LIN {X 0,Y 157.711,Z 411.935,A -85,B 0,C 180,E1 -26136.375,E2 -26136.375} C_VEL
LIN {X 0,Y 161.502,Z 421.422,A -85,B 0,C 180,E1 -26138.842,E2 -26138.842} C_VEL
LIN {X 0,Y 167.93,Z 439.932,A -85,B 0,C 180,E1 -26142.847,E2 -26142.847} C_VEL
LIN {X 0,Y 172.068,Z 451.148,A -85,B 0,C 180,E1 -26145.625,E2 -26145.625} C_VEL
LIN {X 0,Y 176.253,Z 461.302,A -85,B 0,C 180,E1 -26148.517,E2 -26148.517} C_VEL
LIN {X 0,Y 181.026,Z 471.361,A -85,B 0,C 180,E1 -26151.736,E2 -26151.736} C_VEL
LIN {X 0,Y 187.397,Z 481.909,A -85,B 0,C 180,E1 -26155.593,E2 -26155.593} C_VEL
LIN {X 0,Y 193.568,Z 490.168,A -85,B 0,C 180,E1 -26158.913,E2 -26158.913} C_VEL
LIN {X 0,Y 201.708,Z 498.817,A -85,B 0,C 180,E1 -26162.732,E2 -26162.732} C_VEL
LIN {X 0,Y 208.546,Z 504.564,A -85,B 0,C 180,E1 -26165.489,E2 -26165.489} C_VEL
LIN {X 0,Y 218.387,Z 511.229,A -85,B 0,C 180,E1 -26168.946,E2 -26168.946} C_VEL
LIN {X 0,Y 231.636,Z 518.165,A -85,B 0,C 180,E1 -26172.885,E2 -26172.885} C_VEL
LIN {X 0,Y 242.773,Z 523.047,A -85,B 0,C 180,E1 -26175.876,E2 -26175.876} C_VEL
LIN {X 0,Y 253.89,Z 527.504,A -85,B 0,C 180,E1 -26178.827,E2 -26178.827} C_VEL
LIN {X 0,Y 260.167,Z 530.069,A -85,B 0,C 180,E1 -26180.673,E2 -26180.673} C_VEL
LIN {X 0,Y 265.407,Z 532.174,A -85,B 0,C 180,E1 -26182.392,E2 -26182.392} C_VEL
LIN {X 0,Y 269.507,Z 533.855,A -85,B 0,C 180,E1 -26184.013,E2 -26184.013} C_VEL
LIN {X 0,Y 272.328,Z 535.154,A -85,B 0,C 180,E1 -26185.56,E2 -26185.56} C_VEL
LIN {X 0,Y 274.967,Z 536.076,A -85,B 0,C 180,E1 -26187.07,E2 -26187.07} C_VEL
LIN {X 0,Y 276.582,Z 536.626,A -85,B 0,C 180,E1 -26188.544,E2 -26188.544} C_VEL
LIN {X 0,Y 277.498,Z 536.802,A -85,B 0,C 180,E1 -26190,E2 -26190} C_VEL
LIN {X 0,Y 276.603,Z 536.625,A -85,B 0,C 180,E1 -26191.456,E2 -26191.456} C_VEL
LIN {X 0,Y 274.515,Z 535.937,A -85,B 0,C 180,E1 -26193.198,E2 -26193.198} C_VEL
LIN {X 0,Y 272.324,Z 535.154,A -85,B 0,C 180,E1 -26194.44,E2 -26194.44} C_VEL
LIN {X 0,Y 268.7,Z 533.534,A -85,B 0,C 180,E1 -26196.334,E2 -26196.334} C_VEL
LIN {X 0,Y 265.444,Z 532.173,A -85,B 0,C 180,E1 -26197.607,E2 -26197.607} C_VEL
LIN {X 0,Y 260.186,Z 530.068,A -85,B 0,C 180,E1 -26199.327,E2 -26199.327} C_VEL
LIN {X 0,Y 251.348,Z 526.504,A -85,B 0,C 180,E1 -26201.867,E2 -26201.867} C_VEL
LIN {X 0,Y 239.951,Z 521.882,A -85,B 0,C 180,E1 -26204.866,E2 -26204.866} C_VEL
LIN {X 0,Y 226.976,Z 515.933,A -85,B 0,C 180,E1 -26208.439,E2 -26208.439} C_VEL
LIN {X 0,Y 213.38,Z 508.049,A -85,B 0,C 180,E1 -26212.749,E2 -26212.749} C_VEL
LIN {X 0,Y 202.925,Z 499.912,A -85,B 0,C 180,E1 -26216.758,E2 -26216.758} C_VEL
LIN {X 0,Y 195.267,Z 492.096,A -85,B 0,C 180,E1 -26220.256,E2 -26220.256} C_VEL
LIN {X 0,Y 187.81,Z 482.614,A -85,B 0,C 180,E1 -26224.146,E2 -26224.146} C_VEL
LIN {X 0,Y 181.961,Z 473.083,A -85,B 0,C 180,E1 -26227.651,E2 -26227.651} C_VEL
LIN {X 0,Y 177.726,Z 464.648,A -85,B 0,C 180,E1 -26230.43,E2 -26230.43} C_VEL
LIN {X 0,Y 173.629,Z 455.239,A -85,B 0,C 180,E1 -26233.234,E2 -26233.234} C_VEL
LIN {X 0,Y 169.867,Z 445.428,A -85,B 0,C 180,E1 -26235.824,E2 -26235.824} C_VEL
LIN {X 0,Y 166.21,Z 435.07,A -85,B 0,C 180,E1 -26238.245,E2 -26238.245} C_VEL
LIN {X 0,Y 161.21,Z 420.652,A -85,B 0,C 180,E1 -26241.342,E2 -26241.342} C_VEL
LIN {X 0,Y 157.598,Z 411.646,A -85,B 0,C 180,E1 -26243.703,E2 -26243.703} C_VEL
LIN {X 0,Y 153.19,Z 402.471,A -85,B 0,C 180,E1 -26246.795,E2 -26246.795} C_VEL
LIN {X 0,Y 148.612,Z 394.018,A -85,B 0,C 180,E1 -26250.424,E2 -26250.424} C_VEL
LIN {X 0,Y 144.236,Z 386.913,A -85,B 0,C 180,E1 -26254.476,E2 -26254.476} C_VEL
LIN {X 0,Y 141.463,Z 382.764,A -85,B 0,C 180,E1 -26257.501,E2 -26257.501} C_VEL
LIN {X 0,Y 138.857,Z 378.927,A -85,B 0,C 180,E1 -26260.878,E2 -26260.878} C_VEL
LIN {X 0,Y 136.291,Z 375.231,A -85,B 0,C 180,E1 -26265.06,E2 -26265.06} C_VEL
LIN {X 0,Y 135.757,Z 374.279,A -85,B 0,C 180,E1 -26266.149,E2 -26266.149} C_VEL
LIN {X 0,Y 133.455,Z 371.692,A -85,B 0,C 180,E1 -26272.056,E2 -26272.056} C_VEL
LIN {X 0,Y 132.719,Z 369.463,A -85,B 0,C 180,E1 -26276.586,E2 -26276.586} C_VEL
LIN {X 0,Y 132.574,Z 368.941,A -85,B 0,C 180,E1 -26280.002,E2 -26280.002} C_VEL
LIN {X 0,Y 132.851,Z 369.82,A -85,B 0,C 180,E1 -26284.173,E2 -26284.173} C_VEL
LIN {X 0,Y 135.292,Z 374.003,A -85,B 0,C 180,E1 -26292.566,E2 -26292.566} C_VEL
LIN {X 0,Y 136.12,Z 374.835,A -85,B 0,C 180,E1 -26294.198,E2 -26294.198} C_VEL
LIN {X 0,Y 138.416,Z 378.446,A -85,B 0,C 180,E1 -26298.121,E2 -26298.121} C_VEL
LIN {X 0,Y 139.473,Z 379.845,A -85,B 0,C 180,E1 -26299.599,E2 -26299.599} C_VEL
LIN {X 0,Y 142.528,Z 384.331,A -85,B 0,C 180,E1 -26303.331,E2 -26303.331} C_VEL
LIN {X 0,Y 145.453,Z 388.952,A -85,B 0,C 180,E1 -26306.356,E2 -26306.356} C_VEL
LIN {X 0,Y 147.78,Z 392.828,A -85,B 0,C 180,E1 -26308.495,E2 -26308.495} C_VEL
LIN {X 0,Y 151.379,Z 401.147,A -85,B 0,C 180,E1 -26311.635,E2 -26311.635} C_VEL
LIN {X 0,Y 155.437,Z 412.076,A -85,B 0,C 180,E1 -26314.84,E2 -26314.84} C_VEL
LIN {X 0,Y 156.568,Z 415.668,A -85,B 0,C 180,E1 -26315.702,E2 -26315.702} C_VEL
LIN {X 0,Y 154.129,Z 443.65,A -85,B 0,C 180,E1 -26316.777,E2 -26316.777} C_VEL
LIN {X 0,Y 152.023,Z 456.485,A -85,B 0,C 180,E1 -26317.57,E2 -26317.57} C_VEL
LIN {X 0,Y 148.735,Z 469.266,A -85,B 0,C 180,E1 -26318.773,E2 -26318.773} C_VEL
LIN {X 0,Y 145.582,Z 478.774,A -85,B 0,C 180,E1 -26319.973,E2 -26319.973} C_VEL
LIN {X 0,Y 141.897,Z 488.043,A -85,B 0,C 180,E1 -26321.487,E2 -26321.487} C_VEL
LIN {X 0,Y 137.778,Z 496.981,A -85,B 0,C 180,E1 -26323.375,E2 -26323.375} C_VEL
LIN {X 0,Y 133.274,Z 505.504,A -85,B 0,C 180,E1 -26325.677,E2 -26325.677} C_VEL
LIN {X 0,Y 129.051,Z 512.718,A -85,B 0,C 180,E1 -26328.156,E2 -26328.156} C_VEL
LIN {X 0,Y 125.096,Z 518.916,A -85,B 0,C 180,E1 -26330.801,E2 -26330.801} C_VEL
LIN {X 0,Y 120.577,Z 525.451,A -85,B 0,C 180,E1 -26334.349,E2 -26334.349} C_VEL
LIN {X 0,Y 115.984,Z 531.873,A -85,B 0,C 180,E1 -26339,E2 -26339} C_VEL
LIN {X 0,Y 111.97,Z 537.003,A -85,B 0,C 180,E1 -26343.937,E2 -26343.937} C_VEL
LIN {X 0,Y 108.806,Z 540.993,A -85,B 0,C 180,E1 -26349.191,E2 -26349.191} C_VEL
LIN {X 0,Y 106.705,Z 543.952,A -85,B 0,C 180,E1 -26354.725,E2 -26354.725} C_VEL
LIN {X 0,Y 105.264,Z 546.414,A -85,B 0,C 180,E1 -26362.326,E2 -26362.326} C_VEL
LIN {X 0,Y 105.047,Z 547.01,A -85,B 0,C 180,E1 -26366.164,E2 -26366.164} C_VEL
LIN {X 0,Y 105.171,Z 547.172,A -85,B 0,C 180,E1 -26370,E2 -26370} C_VEL
LIN {X 0,Y 105.038,Z 547.01,A -85,B 0,C 180,E1 -26373.836,E2 -26373.836} C_VEL
LIN {X 0,Y 105.226,Z 546.413,A -85,B 0,C 180,E1 -26377.676,E2 -26377.676} C_VEL
LIN {X 0,Y 106.705,Z 543.952,A -85,B 0,C 180,E1 -26385.275,E2 -26385.275} C_VEL
LIN {X 0,Y 108.806,Z 540.993,A -85,B 0,C 180,E1 -26390.809,E2 -26390.809} C_VEL
LIN {X 0,Y 111.97,Z 537.003,A -85,B 0,C 180,E1 -26396.063,E2 -26396.063} C_VEL
LIN {X 0,Y 115.99,Z 531.874,A -85,B 0,C 180,E1 -26400.999,E2 -26400.999} C_VEL
LIN {X 0,Y 120.636,Z 525.453,A -85,B 0,C 180,E1 -26405.631,E2 -26405.631} C_VEL
LIN {X 0,Y 126.046,Z 517.533,A -85,B 0,C 180,E1 -26409.881,E2 -26409.881} C_VEL
LIN {X 0,Y 131.142,Z 509.34,A -85,B 0,C 180,E1 -26413.099,E2 -26413.099} C_VEL
LIN {X 0,Y 136.063,Z 500.383,A -85,B 0,C 180,E1 -26415.78,E2 -26415.78} C_VEL
LIN {X 0,Y 140.126,Z 492.096,A -85,B 0,C 180,E1 -26417.711,E2 -26417.711} C_VEL
LIN {X 0,Y 144.306,Z 482.034,A -85,B 0,C 180,E1 -26419.548,E2 -26419.548} C_VEL
LIN {X 0,Y 147.764,Z 472.284,A -85,B 0,C 180,E1 -26420.881,E2 -26420.881} C_VEL
LIN {X 0,Y 150.284,Z 463.495,A -85,B 0,C 180,E1 -26421.833,E2 -26421.833} C_VEL
LIN {X 0,Y 152.647,Z 453.074,A -85,B 0,C 180,E1 -26422.656,E2 -26422.656} C_VEL
LIN {X 0,Y 154.169,Z 443.105,A -85,B 0,C 180,E1 -26423.25,E2 -26423.25} C_VEL
LIN {X 0,Y 156.565,Z 415.689,A -85,B 0,C 180,E1 -26424.298,E2 -26424.298} C_VEL
LIN {X 0,Y 153.862,Z 407.654,A -85,B 0,C 180,E1 -26426.368,E2 -26426.368} C_VEL
LIN {X 0,Y 149.993,Z 397.773,A -85,B 0,C 180,E1 -26429.538,E2 -26429.538} C_VEL
LIN {X 0,Y 147.077,Z 391.607,A -85,B 0,C 180,E1 -26432.133,E2 -26432.133} C_VEL
LIN {X 0,Y 143.786,Z 386.3,A -85,B 0,C 180,E1 -26435.312,E2 -26435.312} C_VEL
LIN {X 0,Y 141.521,Z 382.829,A -85,B 0,C 180,E1 -26437.819,E2 -26437.819} C_VEL
LIN {X 0,Y 139.084,Z 379.09,A -85,B 0,C 180,E1 -26440.966,E2 -26440.966} C_VEL
LIN {X 0,Y 138.007,Z 378.043,A -85,B 0,C 180,E1 -26442.468,E2 -26442.468} C_VEL
LIN {X 0,Y 136.91,Z 377.653,A -85,B 0,C 180,E1 -26444.037,E2 -26444.037} C_VEL
LIN {X 0,Y 133.217,Z 378.698,A -85,B 0,C 180,E1 -26450.653,E2 -26450.653} C_VEL
LIN {X 0,Y 132.394,Z 378.392,A -85,B 0,C 180,E1 -26453.213,E2 -26453.213} C_VEL
LIN {X 0,Y 132.218,Z 378.001,A -85,B 0,C 180,E1 -26454.058,E2 -26454.058} C_VEL
LIN {X 0,Y 131.788,Z 376.347,A -85,B 0,C 180,E1 -26457.706,E2 -26457.706} C_VEL
LIN {X 0,Y 131.702,Z 376.09,A -85,B 0,C 180,E1 -26460.763,E2 -26460.763} C_VEL
LIN {X 0,Y 131.924,Z 376.857,A -85,B 0,C 180,E1 -26464.199,E2 -26464.199} C_VEL
LIN {X 0,Y 134.158,Z 380.922,A -85,B 0,C 180,E1 -26472.444,E2 -26472.444} C_VEL
LIN {X 0,Y 134.823,Z 381.684,A -85,B 0,C 180,E1 -26473.853,E2 -26473.853} C_VEL
LIN {X 0,Y 137.252,Z 385.481,A -85,B 0,C 180,E1 -26478.181,E2 -26478.181} C_VEL
LIN {X 0,Y 140.462,Z 390.479,A -85,B 0,C 180,E1 -26482.523,E2 -26482.523} C_VEL
LIN {X 0,Y 143.478,Z 395.47,A -85,B 0,C 180,E1 -26485.863,E2 -26485.863} C_VEL
LIN {X 0,Y 147.492,Z 402.492,A -85,B 0,C 180,E1 -26489.626,E2 -26489.626} C_VEL
LIN {X 0,Y 152.1,Z 411.916,A -85,B 0,C 180,E1 -26493.375,E2 -26493.375} C_VEL
LIN {X 0,Y 156.129,Z 421.509,A -85,B 0,C 180,E1 -26496.312,E2 -26496.312} C_VEL
LIN {X 0,Y 159.764,Z 432.052,A -85,B 0,C 180,E1 -26498.817,E2 -26498.817} C_VEL
LIN {X 0,Y 163.355,Z 443.752,A -85,B 0,C 180,E1 -26501.513,E2 -26501.513} C_VEL
LIN {X 0,Y 166.675,Z 453.927,A -85,B 0,C 180,E1 -26504.209,E2 -26504.209} C_VEL
LIN {X 0,Y 170.416,Z 464.042,A -85,B 0,C 180,E1 -26507.268,E2 -26507.268} C_VEL
LIN {X 0,Y 174.817,Z 474.111,A -85,B 0,C 180,E1 -26510.702,E2 -26510.702} C_VEL
LIN {X 0,Y 178.982,Z 481.72,A -85,B 0,C 180,E1 -26513.606,E2 -26513.606} C_VEL
LIN {X 0,Y 184.846,Z 490.495,A -85,B 0,C 180,E1 -26517.285,E2 -26517.285} C_VEL
LIN {X 0,Y 190.862,Z 497.704,A -85,B 0,C 180,E1 -26520.58,E2 -26520.58} C_VEL
LIN {X 0,Y 198.504,Z 504.99,A -85,B 0,C 180,E1 -26524.206,E2 -26524.206} C_VEL
LIN {X 0,Y 208.801,Z 512.388,A -85,B 0,C 180,E1 -26528.27,E2 -26528.27} C_VEL
LIN {X 0,Y 221.304,Z 519.044,A -85,B 0,C 180,E1 -26532.307,E2 -26532.307} C_VEL
LIN {X 0,Y 235.113,Z 524.844,A -85,B 0,C 180,E1 -26536.165,E2 -26536.165} C_VEL
LIN {X 0,Y 246.769,Z 529.058,A -85,B 0,C 180,E1 -26539.279,E2 -26539.279} C_VEL
LIN {X 0,Y 255.571,Z 532.16,A -85,B 0,C 180,E1 -26541.871,E2 -26541.871} C_VEL
LIN {X 0,Y 261.478,Z 534.217,A -85,B 0,C 180,E1 -26543.97,E2 -26543.97} C_VEL
LIN {X 0,Y 264.483,Z 535.367,A -85,B 0,C 180,E1 -26545.428,E2 -26545.428} C_VEL
LIN {X 0,Y 267.412,Z 536.324,A -85,B 0,C 180,E1 -26547.058,E2 -26547.058} C_VEL
LIN {X 0,Y 269.258,Z 536.825,A -85,B 0,C 180,E1 -26548.504,E2 -26548.504} C_VEL
LIN {X 0,Y 270.33,Z 536.994,A -85,B 0,C 180,E1 -26550,E2 -26550} C_VEL
LIN {X 0,Y 269.274,Z 536.824,A -85,B 0,C 180,E1 -26551.496,E2 -26551.496} C_VEL
LIN {X 0,Y 267.267,Z 536.288,A -85,B 0,C 180,E1 -26553.015,E2 -26553.015} C_VEL
LIN {X 0,Y 264.455,Z 535.368,A -85,B 0,C 180,E1 -26554.573,E2 -26554.573} C_VEL
LIN {X 0,Y 261.075,Z 534.088,A -85,B 0,C 180,E1 -26556.181,E2 -26556.181} C_VEL
LIN {X 0,Y 255.574,Z 532.153,A -85,B 0,C 180,E1 -26558.134,E2 -26558.134} C_VEL
LIN {X 0,Y 246.768,Z 529.059,A -85,B 0,C 180,E1 -26560.72,E2 -26560.72} C_VEL
LIN {X 0,Y 235.074,Z 524.846,A -85,B 0,C 180,E1 -26563.838,E2 -26563.838} C_VEL
LIN {X 0,Y 221.304,Z 519.043,A -85,B 0,C 180,E1 -26567.693,E2 -26567.693} C_VEL
LIN {X 0,Y 208.846,Z 512.387,A -85,B 0,C 180,E1 -26571.725,E2 -26571.725} C_VEL
LIN {X 0,Y 200.755,Z 506.782,A -85,B 0,C 180,E1 -26574.84,E2 -26574.84} C_VEL
LIN {X 0,Y 192.265,Z 499.236,A -85,B 0,C 180,E1 -26578.686,E2 -26578.686} C_VEL
LIN {X 0,Y 185.303,Z 491.125,A -85,B 0,C 180,E1 -26582.438,E2 -26582.438} C_VEL
LIN {X 0,Y 179.655,Z 482.876,A -85,B 0,C 180,E1 -26585.929,E2 -26585.929} C_VEL
LIN {X 0,Y 174.806,Z 474.142,A -85,B 0,C 180,E1 -26589.293,E2 -26589.293} C_VEL
LIN {X 0,Y 170.971,Z 465.43,A -85,B 0,C 180,E1 -26592.278,E2 -26592.278} C_VEL
LIN {X 0,Y 168.022,Z 457.733,A -85,B 0,C 180,E1 -26594.68,E2 -26594.68} C_VEL
LIN {X 0,Y 164.732,Z 448.109,A -85,B 0,C 180,E1 -26597.371,E2 -26597.371} C_VEL
LIN {X 0,Y 161.357,Z 437.315,A -85,B 0,C 180,E1 -26600.028,E2 -26600.028} C_VEL
LIN {X 0,Y 157.158,Z 424.418,A -85,B 0,C 180,E1 -26602.959,E2 -26602.959} C_VEL
LIN {X 0,Y 153.804,Z 415.819,A -85,B 0,C 180,E1 -26605.35,E2 -26605.35} C_VEL
LIN {X 0,Y 150.072,Z 407.643,A -85,B 0,C 180,E1 -26608.208,E2 -26608.208} C_VEL
LIN {X 0,Y 146.074,Z 399.864,A -85,B 0,C 180,E1 -26611.642,E2 -26611.642} C_VEL
LIN {X 0,Y 142.005,Z 392.928,A -85,B 0,C 180,E1 -26615.709,E2 -26615.709} C_VEL
LIN {X 0,Y 139.441,Z 388.935,A -85,B 0,C 180,E1 -26618.738,E2 -26618.738} C_VEL
LIN {X 0,Y 137.25,Z 385.508,A -85,B 0,C 180,E1 -26621.817,E2 -26621.817} C_VEL
LIN {X 0,Y 134.783,Z 381.586,A -85,B 0,C 180,E1 -26626.239,E2 -26626.239} C_VEL
LIN {X 0,Y 131.818,Z 376.434,A -85,B 0,C 180,E1 -26636.945,E2 -26636.945} C_VEL
LIN {X 0,Y 131.715,Z 376.082,A -85,B 0,C 180,E1 -26640.766,E2 -26640.766} C_VEL
LIN {X 0,Y 131.953,Z 377.015,A -85,B 0,C 180,E1 -26644.106,E2 -26644.106} C_VEL
LIN {X 0,Y 134.175,Z 380.928,A -85,B 0,C 180,E1 -26652.096,E2 -26652.096} C_VEL
LIN {X 0,Y 134.866,Z 381.77,A -85,B 0,C 180,E1 -26653.564,E2 -26653.564} C_VEL
LIN {X 0,Y 137.314,Z 385.532,A -85,B 0,C 180,E1 -26657.886,E2 -26657.886} C_VEL
LIN {X 0,Y 140.622,Z 390.728,A -85,B 0,C 180,E1 -26662.329,E2 -26662.329} C_VEL
LIN {X 0,Y 144.3,Z 396.751,A -85,B 0,C 180,E1 -26666.291,E2 -26666.291} C_VEL
LIN {X 0,Y 147.272,Z 403.499,A -85,B 0,C 180,E1 -26669.188,E2 -26669.188} C_VEL
LIN {X 0,Y 151.416,Z 414.966,A -85,B 0,C 180,E1 -26672.854,E2 -26672.854} C_VEL
LIN {X 0,Y 152.317,Z 417.977,A -85,B 0,C 180,E1 -26673.622,E2 -26673.622} C_VEL
LIN {X 0,Y 150.023,Z 443.119,A -85,B 0,C 180,E1 -26674.584,E2 -26674.584} C_VEL
LIN {X 0,Y 147.77,Z 456.439,A -85,B 0,C 180,E1 -26675.399,E2 -26675.399} C_VEL
LIN {X 0,Y 144.404,Z 469.072,A -85,B 0,C 180,E1 -26676.581,E2 -26676.581} C_VEL
LIN {X 0,Y 141.129,Z 478.581,A -85,B 0,C 180,E1 -26677.765,E2 -26677.765} C_VEL
LIN {X 0,Y 137.284,Z 487.849,A -85,B 0,C 180,E1 -26679.26,E2 -26679.26} C_VEL
LIN {X 0,Y 133,Z 496.787,A -85,B 0,C 180,E1 -26681.151,E2 -26681.151} C_VEL
LIN {X 0,Y 128.289,Z 505.31,A -85,B 0,C 180,E1 -26683.46,E2 -26683.46} C_VEL
LIN {X 0,Y 123.824,Z 512.523,A -85,B 0,C 180,E1 -26685.951,E2 -26685.951} C_VEL
LIN {X 0,Y 119.659,Z 518.722,A -85,B 0,C 180,E1 -26688.644,E2 -26688.644} C_VEL
LIN {X 0,Y 114.846,Z 525.256,A -85,B 0,C 180,E1 -26692.27,E2 -26692.27} C_VEL
LIN {X 0,Y 109.942,Z 531.679,A -85,B 0,C 180,E1 -26697.088,E2 -26697.088} C_VEL
LIN {X 0,Y 105.604,Z 536.808,A -85,B 0,C 180,E1 -26702.235,E2 -26702.235} C_VEL
LIN {X 0,Y 102.183,Z 540.798,A -85,B 0,C 180,E1 -26707.773,E2 -26707.773} C_VEL
LIN {X 0,Y 99.83,Z 543.757,A -85,B 0,C 180,E1 -26713.645,E2 -26713.645} C_VEL
LIN {X 0,Y 98.213,Z 546.219,A -85,B 0,C 180,E1 -26721.772,E2 -26721.772} C_VEL
LIN {X 0,Y 97.952,Z 546.816,A -85,B 0,C 180,E1 -26725.886,E2 -26725.886} C_VEL
LIN {X 0,Y 98.077,Z 546.978,A -85,B 0,C 180,E1 -26730,E2 -26730} C_VEL
LIN {X 0,Y 97.944,Z 546.816,A -85,B 0,C 180,E1 -26734.115,E2 -26734.115} C_VEL
LIN {X 0,Y 98.183,Z 546.219,A -85,B 0,C 180,E1 -26738.231,E2 -26738.231} C_VEL
LIN {X 0,Y 99.83,Z 543.757,A -85,B 0,C 180,E1 -26746.355,E2 -26746.355} C_VEL
LIN {X 0,Y 102.183,Z 540.798,A -85,B 0,C 180,E1 -26752.227,E2 -26752.227} C_VEL
LIN {X 0,Y 105.603,Z 536.808,A -85,B 0,C 180,E1 -26757.765,E2 -26757.765} C_VEL
LIN {X 0,Y 109.953,Z 531.679,A -85,B 0,C 180,E1 -26762.908,E2 -26762.908} C_VEL
LIN {X 0,Y 114.085,Z 526.335,A -85,B 0,C 180,E1 -26766.99,E2 -26766.99} C_VEL
LIN {X 0,Y 118.657,Z 520.097,A -85,B 0,C 180,E1 -26770.656,E2 -26770.656} C_VEL
LIN {X 0,Y 122.787,Z 514.15,A -85,B 0,C 180,E1 -26773.38,E2 -26773.38} C_VEL
LIN {X 0,Y 127.157,Z 507.228,A -85,B 0,C 180,E1 -26775.93,E2 -26775.93} C_VEL
LIN {X 0,Y 131.789,Z 499.054,A -85,B 0,C 180,E1 -26778.294,E2 -26778.294} C_VEL
LIN {X 0,Y 136.048,Z 490.551,A -85,B 0,C 180,E1 -26780.21,E2 -26780.21} C_VEL
LIN {X 0,Y 139.798,Z 481.84,A -85,B 0,C 180,E1 -26781.766,E2 -26781.766} C_VEL
LIN {X 0,Y 143.402,Z 472.091,A -85,B 0,C 180,E1 -26783.077,E2 -26783.077} C_VEL
LIN {X 0,Y 146.337,Z 462.014,A -85,B 0,C 180,E1 -26784.137,E2 -26784.137} C_VEL
LIN {X 0,Y 148.531,Z 452.364,A -85,B 0,C 180,E1 -26784.876,E2 -26784.876} C_VEL
LIN {X 0,Y 150.194,Z 441.64,A -85,B 0,C 180,E1 -26785.472,E2 -26785.472} C_VEL
LIN {X 0,Y 152.312,Z 418.029,A -85,B 0,C 180,E1 -26786.377,E2 -26786.377} C_VEL
LIN {X 0,Y 150.046,Z 411.134,A -85,B 0,C 180,E1 -26788.298,E2 -26788.298} C_VEL
LIN {X 0,Y 146.678,Z 402.068,A -85,B 0,C 180,E1 -26791.369,E2 -26791.369} C_VEL
LIN {X 0,Y 144.214,Z 396.644,A -85,B 0,C 180,E1 -26793.79,E2 -26793.79} C_VEL
LIN {X 0,Y 141.079,Z 391.529,A -85,B 0,C 180,E1 -26797.126,E2 -26797.126} C_VEL
LIN {X 0,Y 139.562,Z 389.099,A -85,B 0,C 180,E1 -26798.971,E2 -26798.971} C_VEL
LIN {X 0,Y 137.077,Z 385.251,A -85,B 0,C 180,E1 -26802.468,E2 -26802.468} C_VEL
LIN {X 0,Y 134.783,Z 381.598,A -85,B 0,C 180,E1 -26806.62,E2 -26806.62} C_VEL
LIN {X 0,Y 132.218,Z 378.001,A -85,B 0,C 180,E1 -26814.058,E2 -26814.058} C_VEL
LIN {X 0,Y 131.915,Z 377.541,A -85,B 0,C 180,E1 -26815.739,E2 -26815.739} C_VEL
LIN {X 0,Y 131.628,Z 377.878,A -85,B 0,C 180,E1 -26817.437,E2 -26817.437} C_VEL
LIN {X 0,Y 131.289,Z 379.409,A -85,B 0,C 180,E1 -26819.952,E2 -26819.952} C_VEL
LIN {X 0,Y 131.267,Z 384.714,A -85,B 0,C 180,E1 -26825.809,E2 -26825.809} C_VEL
LIN {X 0,Y 131.579,Z 385.831,A -85,B 0,C 180,E1 -26827.537,E2 -26827.537} C_VEL
LIN {X 0,Y 133.476,Z 388.337,A -85,B 0,C 180,E1 -26832.929,E2 -26832.929} C_VEL
LIN {X 0,Y 136.352,Z 393.196,A -85,B 0,C 180,E1 -26838.305,E2 -26838.305} C_VEL
LIN {X 0,Y 138.762,Z 397.166,A -85,B 0,C 180,E1 -26841.69,E2 -26841.69} C_VEL
LIN {X 0,Y 142.109,Z 402.924,A -85,B 0,C 180,E1 -26845.565,E2 -26845.565} C_VEL
LIN {X 0,Y 145.99,Z 410.51,A -85,B 0,C 180,E1 -26849.367,E2 -26849.367} C_VEL
LIN {X 0,Y 149.899,Z 419.269,A -85,B 0,C 180,E1 -26852.714,E2 -26852.714} C_VEL
LIN {X 0,Y 153.319,Z 428.275,A -85,B 0,C 180,E1 -26855.39,E2 -26855.39} C_VEL
LIN {X 0,Y 156.443,Z 438.884,A -85,B 0,C 180,E1 -26857.942,E2 -26857.942} C_VEL
LIN {X 0,Y 159.898,Z 451.346,A -85,B 0,C 180,E1 -26861.14,E2 -26861.14} C_VEL
LIN {X 0,Y 163.516,Z 463.236,A -85,B 0,C 180,E1 -26864.759,E2 -26864.759} C_VEL
LIN {X 0,Y 167.152,Z 473.109,A -85,B 0,C 180,E1 -26868.2,E2 -26868.2} C_VEL
LIN {X 0,Y 170.845,Z 481.411,A -85,B 0,C 180,E1 -26871.405,E2 -26871.405} C_VEL
LIN {X 0,Y 176.44,Z 490.914,A -85,B 0,C 180,E1 -26875.561,E2 -26875.561} C_VEL
LIN {X 0,Y 183.13,Z 499.591,A -85,B 0,C 180,E1 -26879.765,E2 -26879.765} C_VEL
LIN {X 0,Y 190.675,Z 507.079,A -85,B 0,C 180,E1 -26883.75,E2 -26883.75} C_VEL
LIN {X 0,Y 200.766,Z 514.405,A -85,B 0,C 180,E1 -26888.069,E2 -26888.069} C_VEL
LIN {X 0,Y 214.865,Z 521.668,A -85,B 0,C 180,E1 -26892.88,E2 -26892.88} C_VEL
LIN {X 0,Y 224.763,Z 525.598,A -85,B 0,C 180,E1 -26895.767,E2 -26895.767} C_VEL
LIN {X 0,Y 236.331,Z 529.518,A -85,B 0,C 180,E1 -26898.912,E2 -26898.912} C_VEL
LIN {X 0,Y 242.263,Z 531.309,A -85,B 0,C 180,E1 -26900.509,E2 -26900.509} C_VEL
LIN {X 0,Y 248.225,Z 533.13,A -85,B 0,C 180,E1 -26902.281,E2 -26902.281} C_VEL
LIN {X 0,Y 254.246,Z 534.932,A -85,B 0,C 180,E1 -26904.332,E2 -26904.332} C_VEL
LIN {X 0,Y 256.411,Z 535.586,A -85,B 0,C 180,E1 -26905.284,E2 -26905.284} C_VEL
LIN {X 0,Y 260.312,Z 536.689,A -85,B 0,C 180,E1 -26907.337,E2 -26907.337} C_VEL
LIN {X 0,Y 261.839,Z 537.027,A -85,B 0,C 180,E1 -26908.462,E2 -26908.462} C_VEL
LIN {X 0,Y 263.138,Z 537.187,A -85,B 0,C 180,E1 -26910,E2 -26910} C_VEL
LIN {X 0,Y 261.85,Z 537.026,A -85,B 0,C 180,E1 -26911.538,E2 -26911.538} C_VEL
LIN {X 0,Y 259.497,Z 536.502,A -85,B 0,C 180,E1 -26913.105,E2 -26913.105} C_VEL
LIN {X 0,Y 256.384,Z 535.587,A -85,B 0,C 180,E1 -26914.717,E2 -26914.717} C_VEL
LIN {X 0,Y 254.247,Z 534.932,A -85,B 0,C 180,E1 -26915.669,E2 -26915.669} C_VEL
LIN {X 0,Y 248.226,Z 533.127,A -85,B 0,C 180,E1 -26917.722,E2 -26917.722} C_VEL
LIN {X 0,Y 239.939,Z 530.619,A -85,B 0,C 180,E1 -26920.122,E2 -26920.122} C_VEL
LIN {X 0,Y 230.494,Z 527.587,A -85,B 0,C 180,E1 -26922.659,E2 -26922.659} C_VEL
LIN {X 0,Y 219.142,Z 523.426,A -85,B 0,C 180,E1 -26925.826,E2 -26925.826} C_VEL
LIN {X 0,Y 206.25,Z 517.519,A -85,B 0,C 180,E1 -26929.922,E2 -26929.922} C_VEL
LIN {X 0,Y 196.308,Z 511.419,A -85,B 0,C 180,E1 -26933.742,E2 -26933.742} C_VEL
LIN {X 0,Y 187.126,Z 503.852,A -85,B 0,C 180,E1 -26938.045,E2 -26938.045} C_VEL
LIN {X 0,Y 179.289,Z 494.956,A -85,B 0,C 180,E1 -26942.57,E2 -26942.57} C_VEL
LIN {X 0,Y 173.217,Z 485.793,A -85,B 0,C 180,E1 -26946.746,E2 -26946.746} C_VEL
LIN {X 0,Y 168.495,Z 476.501,A -85,B 0,C 180,E1 -26950.547,E2 -26950.547} C_VEL
LIN {X 0,Y 165.15,Z 467.894,A -85,B 0,C 180,E1 -26953.663,E2 -26953.663} C_VEL
LIN {X 0,Y 162.046,Z 458.734,A -85,B 0,C 180,E1 -26956.672,E2 -26956.672} C_VEL
LIN {X 0,Y 158.955,Z 448.136,A -85,B 0,C 180,E1 -26959.714,E2 -26959.714} C_VEL
LIN {X 0,Y 156.21,Z 437.899,A -85,B 0,C 180,E1 -26962.297,E2 -26962.297} C_VEL
LIN {X 0,Y 152.902,Z 427.096,A -85,B 0,C 180,E1 -26964.927,E2 -26964.927} C_VEL
LIN {X 0,Y 149.498,Z 418.281,A -85,B 0,C 180,E1 -26967.616,E2 -26967.616} C_VEL
LIN {X 0,Y 145.465,Z 409.458,A -85,B 0,C 180,E1 -26971.111,E2 -26971.111} C_VEL
LIN {X 0,Y 141.814,Z 402.426,A -85,B 0,C 180,E1 -26974.746,E2 -26974.746} C_VEL
LIN {X 0,Y 138.144,Z 395.984,A -85,B 0,C 180,E1 -26979.14,E2 -26979.14} C_VEL
LIN {X 0,Y 135.574,Z 391.947,A -85,B 0,C 180,E1 -26982.951,E2 -26982.951} C_VEL
LIN {X 0,Y 133.305,Z 388.029,A -85,B 0,C 180,E1 -26987.476,E2 -26987.476} C_VEL
LIN {X 0,Y 131.171,Z 384.732,A -85,B 0,C 180,E1 -26994.622,E2 -26994.622} C_VEL
LIN {X 0,Y 130.892,Z 383.363,A -85,B 0,C 180,E1 -26997.694,E2 -26997.694} C_VEL
LIN {X 0,Y 130.848,Z 383.143,A -85,B 0,C 180,E1 -27000.771,E2 -27000.771} C_VEL
LIN {X 0,Y 131.021,Z 383.988,A -85,B 0,C 180,E1 -27003.654,E2 -27003.654} C_VEL
LIN {X 0,Y 133.15,Z 387.922,A -85,B 0,C 180,E1 -27011.804,E2 -27011.804} C_VEL
LIN {X 0,Y 133.689,Z 388.831,A -85,B 0,C 180,E1 -27013.057,E2 -27013.057} C_VEL
LIN {X 0,Y 136.238,Z 392.995,A -85,B 0,C 180,E1 -27017.741,E2 -27017.741} C_VEL
LIN {X 0,Y 138.73,Z 397.061,A -85,B 0,C 180,E1 -27021.259,E2 -27021.259} C_VEL
LIN {X 0,Y 142.07,Z 402.906,A -85,B 0,C 180,E1 -27025.146,E2 -27025.146} C_VEL
LIN {X 0,Y 144.479,Z 408.888,A -85,B 0,C 180,E1 -27027.722,E2 -27027.722} C_VEL
LIN {X 0,Y 148.195,Z 420.105,A -85,B 0,C 180,E1 -27031.356,E2 -27031.356} C_VEL
LIN {X 0,Y 148.316,Z 420.517,A -85,B 0,C 180,E1 -27031.47,E2 -27031.47} C_VEL
LIN {X 0,Y 146.02,Z 443.669,A -85,B 0,C 180,E1 -27032.33,E2 -27032.33} C_VEL
LIN {X 0,Y 143.407,Z 457.785,A -85,B 0,C 180,E1 -27033.219,E2 -27033.219} C_VEL
LIN {X 0,Y 140.297,Z 468.879,A -85,B 0,C 180,E1 -27034.256,E2 -27034.256} C_VEL
LIN {X 0,Y 136.894,Z 478.387,A -85,B 0,C 180,E1 -27035.414,E2 -27035.414} C_VEL
LIN {X 0,Y 132.911,Z 487.655,A -85,B 0,C 180,E1 -27036.893,E2 -27036.893} C_VEL
LIN {X 0,Y 128.437,Z 496.593,A -85,B 0,C 180,E1 -27038.764,E2 -27038.764} C_VEL
LIN {X 0,Y 123.512,Z 505.116,A -85,B 0,C 180,E1 -27041.069,E2 -27041.069} C_VEL
LIN {X 0,Y 118.809,Z 512.329,A -85,B 0,C 180,E1 -27043.563,E2 -27043.563} C_VEL
LIN {X 0,Y 114.397,Z 518.527,A -85,B 0,C 180,E1 -27046.28,E2 -27046.28} C_VEL
LIN {X 0,Y 109.293,Z 525.061,A -85,B 0,C 180,E1 -27049.982,E2 -27049.982} C_VEL
LIN {X 0,Y 105.698,Z 529.566,A -85,B 0,C 180,E1 -27053.244,E2 -27053.244} C_VEL
LIN {X 0,Y 100.764,Z 535.058,A -85,B 0,C 180,E1 -27058.46,E2 -27058.46} C_VEL
LIN {X 0,Y 96.764,Z 539.386,A -85,B 0,C 180,E1 -27064.166,E2 -27064.166} C_VEL
LIN {X 0,Y 94.595,Z 541.756,A -85,B 0,C 180,E1 -27068.194,E2 -27068.194} C_VEL
LIN {X 0,Y 93.005,Z 543.562,A -85,B 0,C 180,E1 -27072.407,E2 -27072.407} C_VEL
LIN {X 0,Y 91.167,Z 546.025,A -85,B 0,C 180,E1 -27081.131,E2 -27081.131} C_VEL
LIN {X 0,Y 90.881,Z 546.622,A -85,B 0,C 180,E1 -27085.565,E2 -27085.565} C_VEL
LIN {X 0,Y 90.976,Z 546.785,A -85,B 0,C 180,E1 -27090,E2 -27090} C_VEL
LIN {X 0,Y 90.873,Z 546.622,A -85,B 0,C 180,E1 -27094.435,E2 -27094.435} C_VEL
LIN {X 0,Y 91.143,Z 546.024,A -85,B 0,C 180,E1 -27098.871,E2 -27098.871} C_VEL
LIN {X 0,Y 93.004,Z 543.562,A -85,B 0,C 180,E1 -27107.593,E2 -27107.593} C_VEL
LIN {X 0,Y 95.61,Z 540.603,A -85,B 0,C 180,E1 -27113.846,E2 -27113.846} C_VEL
LIN {X 0,Y 99.332,Z 536.613,A -85,B 0,C 180,E1 -27119.687,E2 -27119.687} C_VEL
LIN {X 0,Y 104.03,Z 531.484,A -85,B 0,C 180,E1 -27125.045,E2 -27125.045} C_VEL
LIN {X 0,Y 109.356,Z 525.064,A -85,B 0,C 180,E1 -27129.99,E2 -27129.99} C_VEL
LIN {X 0,Y 115.494,Z 517.145,A -85,B 0,C 180,E1 -27134.409,E2 -27134.409} C_VEL
LIN {X 0,Y 121.143,Z 508.952,A -85,B 0,C 180,E1 -27137.702,E2 -27137.702} C_VEL
LIN {X 0,Y 126.56,Z 499.995,A -85,B 0,C 180,E1 -27140.397,E2 -27140.397} C_VEL
LIN {X 0,Y 130.968,Z 491.707,A -85,B 0,C 180,E1 -27142.326,E2 -27142.326} C_VEL
LIN {X 0,Y 135.517,Z 481.646,A -85,B 0,C 180,E1 -27144.126,E2 -27144.126} C_VEL
LIN {X 0,Y 139.254,Z 471.897,A -85,B 0,C 180,E1 -27145.412,E2 -27145.412} C_VEL
LIN {X 0,Y 142.294,Z 461.82,A -85,B 0,C 180,E1 -27146.454,E2 -27146.454} C_VEL
LIN {X 0,Y 144.681,Z 451.565,A -85,B 0,C 180,E1 -27147.217,E2 -27147.217} C_VEL
LIN {X 0,Y 146.278,Z 441.46,A -85,B 0,C 180,E1 -27147.768,E2 -27147.768} C_VEL
LIN {X 0,Y 148.269,Z 420.379,A -85,B 0,C 180,E1 -27148.572,E2 -27148.572} C_VEL
LIN {X 0,Y 145.43,Z 411.686,A -85,B 0,C 180,E1 -27151.297,E2 -27151.297} C_VEL
LIN {X 0,Y 142.995,Z 405.058,A -85,B 0,C 180,E1 -27153.843,E2 -27153.843} C_VEL
LIN {X 0,Y 141.152,Z 401.329,A -85,B 0,C 180,E1 -27155.843,E2 -27155.843} C_VEL
LIN {X 0,Y 138.008,Z 395.807,A -85,B 0,C 180,E1 -27159.699,E2 -27159.699} C_VEL
LIN {X 0,Y 135.522,Z 391.848,A -85,B 0,C 180,E1 -27163.426,E2 -27163.426} C_VEL
LIN {X 0,Y 133.319,Z 388.058,A -85,B 0,C 180,E1 -27167.825,E2 -27167.825} C_VEL
LIN {X 0,Y 131.126,Z 384.484,A -85,B 0,C 180,E1 -27175.387,E2 -27175.387} C_VEL
LIN {X 0,Y 130.919,Z 383.429,A -85,B 0,C 180,E1 -27177.691,E2 -27177.691} C_VEL
LIN {X 0,Y 130.842,Z 383.046,A -85,B 0,C 180,E1 -27179.998,E2 -27179.998} C_VEL
LIN {X 0,Y 131.005,Z 383.88,A -85,B 0,C 180,E1 -27183.843,E2 -27183.843} C_VEL
LIN {X 0,Y 131.579,Z 385.831,A -85,B 0,C 180,E1 -27187.537,E2 -27187.537} C_VEL
LIN {X 0,Y 132.161,Z 387.834,A -85,B 0,C 180,E1 -27189.937,E2 -27189.937} C_VEL
LIN {X 0,Y 132.758,Z 390.863,A -85,B 0,C 180,E1 -27192.14,E2 -27192.14} C_VEL
LIN {X 0,Y 134.279,Z 397.908,A -85,B 0,C 180,E1 -27196.286,E2 -27196.286} C_VEL
LIN {X 0,Y 135.452,Z 400.943,A -85,B 0,C 180,E1 -27198.434,E2 -27198.434} C_VEL
LIN {X 0,Y 135.942,Z 401.753,A -85,B 0,C 180,E1 -27199.18,E2 -27199.18} C_VEL
LIN {X 0,Y 138.912,Z 407.173,A -85,B 0,C 180,E1 -27203.182,E2 -27203.182} C_VEL
LIN {X 0,Y 142.201,Z 413.624,A -85,B 0,C 180,E1 -27206.848,E2 -27206.848} C_VEL
LIN {X 0,Y 146.109,Z 422.64,A -85,B 0,C 180,E1 -27210.624,E2 -27210.624} C_VEL
LIN {X 0,Y 149.274,Z 431.268,A -85,B 0,C 180,E1 -27213.383,E2 -27213.383} C_VEL
LIN {X 0,Y 152.037,Z 441.4,A -85,B 0,C 180,E1 -27216.009,E2 -27216.009} C_VEL
LIN {X 0,Y 154.664,Z 452.736,A -85,B 0,C 180,E1 -27219.084,E2 -27219.084} C_VEL
LIN {X 0,Y 157.409,Z 463.723,A -85,B 0,C 180,E1 -27222.529,E2 -27222.529} C_VEL
LIN {X 0,Y 160.126,Z 472.787,A -85,B 0,C 180,E1 -27225.753,E2 -27225.753} C_VEL
LIN {X 0,Y 163.842,Z 482.557,A -85,B 0,C 180,E1 -27229.698,E2 -27229.698} C_VEL
LIN {X 0,Y 168.316,Z 491.246,A -85,B 0,C 180,E1 -27233.665,E2 -27233.665} C_VEL
LIN {X 0,Y 173.012,Z 498.314,A -85,B 0,C 180,E1 -27237.209,E2 -27237.209} C_VEL
LIN {X 0,Y 179.291,Z 505.618,A -85,B 0,C 180,E1 -27241.221,E2 -27241.221} C_VEL
LIN {X 0,Y 186.221,Z 511.799,A -85,B 0,C 180,E1 -27244.923,E2 -27244.923} C_VEL
LIN {X 0,Y 195.653,Z 518.039,A -85,B 0,C 180,E1 -27249.054,E2 -27249.054} C_VEL
LIN {X 0,Y 206.024,Z 523.12,A -85,B 0,C 180,E1 -27252.771,E2 -27252.771} C_VEL
LIN {X 0,Y 217.149,Z 527.318,A -85,B 0,C 180,E1 -27256.15,E2 -27256.15} C_VEL
LIN {X 0,Y 228.898,Z 530.919,A -85,B 0,C 180,E1 -27259.384,E2 -27259.384} C_VEL
LIN {X 0,Y 236.615,Z 532.968,A -85,B 0,C 180,E1 -27261.46,E2 -27261.46} C_VEL
LIN {X 0,Y 242.954,Z 534.588,A -85,B 0,C 180,E1 -27263.356,E2 -27263.356} C_VEL
LIN {X 0,Y 248.105,Z 535.812,A -85,B 0,C 180,E1 -27265.125,E2 -27265.125} C_VEL
LIN {X 0,Y 253.218,Z 537.016,A -85,B 0,C 180,E1 -27267.644,E2 -27267.644} C_VEL
LIN {X 0,Y 254.357,Z 537.23,A -85,B 0,C 180,E1 -27268.417,E2 -27268.417} C_VEL
LIN {X 0,Y 255.915,Z 537.38,A -85,B 0,C 180,E1 -27270,E2 -27270} C_VEL
LIN {X 0,Y 254.353,Z 537.23,A -85,B 0,C 180,E1 -27271.583,E2 -27271.583} C_VEL
LIN {X 0,Y 251.57,Z 536.72,A -85,B 0,C 180,E1 -27273.203,E2 -27273.203} C_VEL
LIN {X 0,Y 248.104,Z 535.812,A -85,B 0,C 180,E1 -27274.875,E2 -27274.875} C_VEL
LIN {X 0,Y 242.964,Z 534.588,A -85,B 0,C 180,E1 -27276.644,E2 -27276.644} C_VEL
LIN {X 0,Y 234.825,Z 532.515,A -85,B 0,C 180,E1 -27279.022,E2 -27279.022} C_VEL
LIN {X 0,Y 222.924,Z 529.195,A -85,B 0,C 180,E1 -27282.232,E2 -27282.232} C_VEL
LIN {X 0,Y 208.747,Z 524.228,A -85,B 0,C 180,E1 -27286.362,E2 -27286.362} C_VEL
LIN {X 0,Y 198.171,Z 519.394,A -85,B 0,C 180,E1 -27289.985,E2 -27289.985} C_VEL
LIN {X 0,Y 187.857,Z 512.995,A -85,B 0,C 180,E1 -27294.3,E2 -27294.3} C_VEL
LIN {X 0,Y 181.017,Z 507.366,A -85,B 0,C 180,E1 -27297.768,E2 -27297.768} C_VEL
LIN {X 0,Y 174.083,Z 499.754,A -85,B 0,C 180,E1 -27302.029,E2 -27302.029} C_VEL
LIN {X 0,Y 169.272,Z 492.912,A -85,B 0,C 180,E1 -27305.539,E2 -27305.539} C_VEL
LIN {X 0,Y 165.157,Z 485.422,A -85,B 0,C 180,E1 -27309.052,E2 -27309.052} C_VEL
LIN {X 0,Y 161.81,Z 477.479,A -85,B 0,C 180,E1 -27312.409,E2 -27312.409} C_VEL
LIN {X 0,Y 158.953,Z 469.11,A -85,B 0,C 180,E1 -27315.611,E2 -27315.611} C_VEL
LIN {X 0,Y 156.251,Z 459.513,A -85,B 0,C 180,E1 -27318.87,E2 -27318.87} C_VEL
LIN {X 0,Y 153.55,Z 448.397,A -85,B 0,C 180,E1 -27322.151,E2 -27322.151} C_VEL
LIN {X 0,Y 150.924,Z 436.9,A -85,B 0,C 180,E1 -27325.119,E2 -27325.119} C_VEL
LIN {X 0,Y 147.838,Z 427.104,A -85,B 0,C 180,E1 -27327.85,E2 -27327.85} C_VEL
LIN {X 0,Y 144.288,Z 418.313,A -85,B 0,C 180,E1 -27331.066,E2 -27331.066} C_VEL
LIN {X 0,Y 140.985,Z 411.164,A -85,B 0,C 180,E1 -27334.439,E2 -27334.439} C_VEL
LIN {X 0,Y 137.689,Z 404.876,A -85,B 0,C 180,E1 -27338.368,E2 -27338.368} C_VEL
LIN {X 0,Y 135.712,Z 401.408,A -85,B 0,C 180,E1 -27341.16,E2 -27341.16} C_VEL
LIN {X 0,Y 134.008,Z 398.432,A -85,B 0,C 180,E1 -27344.02,E2 -27344.02} C_VEL
LIN {X 0,Y 131.978,Z 394.776,A -85,B 0,C 180,E1 -27348.468,E2 -27348.468} C_VEL
LIN {X 0,Y 130.135,Z 391.217,A -85,B 0,C 180,E1 -27355.937,E2 -27355.937} C_VEL
LIN {X 0,Y 130.023,Z 390.441,A -85,B 0,C 180,E1 -27357.678,E2 -27357.678} C_VEL
LIN {X 0,Y 129.983,Z 390.186,A -85,B 0,C 180,E1 -27360.776,E2 -27360.776} C_VEL
LIN {X 0,Y 130.119,Z 391.115,A -85,B 0,C 180,E1 -27363.485,E2 -27363.485} C_VEL
LIN {X 0,Y 132.271,Z 395.24,A -85,B 0,C 180,E1 -27371.883,E2 -27371.883} C_VEL
LIN {X 0,Y 134.72,Z 399.649,A -85,B 0,C 180,E1 -27376.853,E2 -27376.853} C_VEL
LIN {X 0,Y 136.836,Z 403.326,A -85,B 0,C 180,E1 -27380.09,E2 -27380.09} C_VEL
LIN {X 0,Y 139.852,Z 408.908,A -85,B 0,C 180,E1 -27383.903,E2 -27383.903} C_VEL
LIN {X 0,Y 142.257,Z 415.801,A -85,B 0,C 180,E1 -27386.748,E2 -27386.748} C_VEL
LIN {X 0,Y 144.445,Z 422.837,A -85,B 0,C 180,E1 -27389.116,E2 -27389.116} C_VEL
LIN {X 0,Y 142.308,Z 443.759,A -85,B 0,C 180,E1 -27389.924,E2 -27389.924} C_VEL
LIN {X 0,Y 139.758,Z 457.165,A -85,B 0,C 180,E1 -27390.745,E2 -27390.745} C_VEL
LIN {X 0,Y 136.432,Z 468.685,A -85,B 0,C 180,E1 -27391.795,E2 -27391.795} C_VEL
LIN {X 0,Y 132.896,Z 478.192,A -85,B 0,C 180,E1 -27392.912,E2 -27392.912} C_VEL
LIN {X 0,Y 128.78,Z 487.462,A -85,B 0,C 180,E1 -27394.37,E2 -27394.37} C_VEL
LIN {X 0,Y 124.116,Z 496.4,A -85,B 0,C 180,E1 -27396.208,E2 -27396.208} C_VEL
LIN {X 0,Y 118.955,Z 504.921,A -85,B 0,C 180,E1 -27398.482,E2 -27398.482} C_VEL
LIN {X 0,Y 114.028,Z 512.135,A -85,B 0,C 180,E1 -27400.975,E2 -27400.975} C_VEL
LIN {X 0,Y 109.364,Z 518.332,A -85,B 0,C 180,E1 -27403.703,E2 -27403.703} C_VEL
LIN {X 0,Y 103.932,Z 524.867,A -85,B 0,C 180,E1 -27407.453,E2 -27407.453} C_VEL
LIN {X 0,Y 100.044,Z 529.371,A -85,B 0,C 180,E1 -27410.785,E2 -27410.785} C_VEL
LIN {X 0,Y 94.764,Z 534.863,A -85,B 0,C 180,E1 -27416.206,E2 -27416.206} C_VEL
LIN {X 0,Y 90.391,Z 539.191,A -85,B 0,C 180,E1 -27422.193,E2 -27422.193} C_VEL
LIN {X 0,Y 88.006,Z 541.561,A -85,B 0,C 180,E1 -27426.467,E2 -27426.467} C_VEL
LIN {X 0,Y 86.238,Z 543.367,A -85,B 0,C 180,E1 -27430.975,E2 -27430.975} C_VEL
LIN {X 0,Y 84.149,Z 545.831,A -85,B 0,C 180,E1 -27440.385,E2 -27440.385} C_VEL
LIN {X 0,Y 83.796,Z 546.428,A -85,B 0,C 180,E1 -27445.189,E2 -27445.189} C_VEL
LIN {X 0,Y 83.883,Z 546.591,A -85,B 0,C 180,E1 -27450,E2 -27450} C_VEL
LIN {X 0,Y 83.79,Z 546.428,A -85,B 0,C 180,E1 -27454.811,E2 -27454.811} C_VEL
LIN {X 0,Y 84.13,Z 545.83,A -85,B 0,C 180,E1 -27459.618,E2 -27459.618} C_VEL
LIN {X 0,Y 86.237,Z 543.367,A -85,B 0,C 180,E1 -27469.025,E2 -27469.025} C_VEL
LIN {X 0,Y 89.135,Z 540.409,A -85,B 0,C 180,E1 -27475.699,E2 -27475.699} C_VEL
LIN {X 0,Y 93.19,Z 536.417,A -85,B 0,C 180,E1 -27481.863,E2 -27481.863} C_VEL
LIN {X 0,Y 98.269,Z 531.289,A -85,B 0,C 180,E1 -27487.437,E2 -27487.437} C_VEL
LIN {X 0,Y 102.997,Z 526.01,A -85,B 0,C 180,E1 -27491.719,E2 -27491.719} C_VEL
LIN {X 0,Y 108.243,Z 519.708,A -85,B 0,C 180,E1 -27495.577,E2 -27495.577} C_VEL
LIN {X 0,Y 112.851,Z 513.761,A -85,B 0,C 180,E1 -27498.357,E2 -27498.357} C_VEL
LIN {X 0,Y 117.715,Z 506.84,A -85,B 0,C 180,E1 -27500.907,E2 -27500.907} C_VEL
LIN {X 0,Y 122.795,Z 498.666,A -85,B 0,C 180,E1 -27503.25,E2 -27503.25} C_VEL
LIN {X 0,Y 127.431,Z 490.163,A -85,B 0,C 180,E1 -27505.12,E2 -27505.12} C_VEL
LIN {X 0,Y 131.487,Z 481.453,A -85,B 0,C 180,E1 -27506.63,E2 -27506.63} C_VEL
LIN {X 0,Y 135.357,Z 471.703,A -85,B 0,C 180,E1 -27507.882,E2 -27507.882} C_VEL
LIN {X 0,Y 138.494,Z 461.626,A -85,B 0,C 180,E1 -27508.905,E2 -27508.905} C_VEL
LIN {X 0,Y 140.99,Z 451.278,A -85,B 0,C 180,E1 -27509.644,E2 -27509.644} C_VEL
LIN {X 0,Y 142.613,Z 441.29,A -85,B 0,C 180,E1 -27510.181,E2 -27510.181} C_VEL
LIN {X 0,Y 144.448,Z 422.809,A -85,B 0,C 180,E1 -27510.885,E2 -27510.885} C_VEL
LIN {X 0,Y 141.183,Z 412.544,A -85,B 0,C 180,E1 -27514.495,E2 -27514.495} C_VEL
LIN {X 0,Y 139.408,Z 408.061,A -85,B 0,C 180,E1 -27516.614,E2 -27516.614} C_VEL
LIN {X 0,Y 136.255,Z 402.223,A -85,B 0,C 180,E1 -27520.752,E2 -27520.752} C_VEL
LIN {X 0,Y 134.012,Z 398.386,A -85,B 0,C 180,E1 -27524.407,E2 -27524.407} C_VEL
LIN {X 0,Y 131.972,Z 394.759,A -85,B 0,C 180,E1 -27528.868,E2 -27528.868} C_VEL
LIN {X 0,Y 130.007,Z 390.333,A -85,B 0,C 180,E1 -27538.449,E2 -27538.449} C_VEL
LIN {X 0,Y 129.97,Z 390.196,A -85,B 0,C 180,E1 -27540.773,E2 -27540.773} C_VEL
LIN {X 0,Y 130.105,Z 391.001,A -85,B 0,C 180,E1 -27543.676,E2 -27543.676} C_VEL
LIN {X 0,Y 131.976,Z 394.788,A -85,B 0,C 180,E1 -27551.532,E2 -27551.532} C_VEL
LIN {X 0,Y 134.681,Z 399.55,A -85,B 0,C 180,E1 -27557.165,E2 -27557.165} C_VEL
LIN {X 0,Y 135.942,Z 401.753,A -85,B 0,C 180,E1 -27559.18,E2 -27559.18} C_VEL
LIN {X 0,Y 136.884,Z 403.609,A -85,B 0,C 180,E1 -27560.571,E2 -27560.571} C_VEL
LIN {X 0,Y 138.05,Z 407.482,A -85,B 0,C 180,E1 -27562.365,E2 -27562.365} C_VEL
LIN {X 0,Y 138.997,Z 412.076,A -85,B 0,C 180,E1 -27563.89,E2 -27563.89} C_VEL
LIN {X 0,Y 141.011,Z 421.868,A -85,B 0,C 180,E1 -27566.802,E2 -27566.802} C_VEL
LIN {X 0,Y 141.98,Z 424.784,A -85,B 0,C 180,E1 -27567.884,E2 -27567.884} C_VEL
LIN {X 0,Y 145.006,Z 433.052,A -85,B 0,C 180,E1 -27570.892,E2 -27570.892} C_VEL
LIN {X 0,Y 147.598,Z 443.22,A -85,B 0,C 180,E1 -27573.813,E2 -27573.813} C_VEL
LIN {X 0,Y 149.662,Z 454.639,A -85,B 0,C 180,E1 -27577.033,E2 -27577.033} C_VEL
LIN {X 0,Y 151.536,Z 463.866,A -85,B 0,C 180,E1 -27580.023,E2 -27580.023} C_VEL
LIN {X 0,Y 153.687,Z 472.843,A -85,B 0,C 180,E1 -27583.307,E2 -27583.307} C_VEL
LIN {X 0,Y 156.453,Z 481.798,A -85,B 0,C 180,E1 -27587.022,E2 -27587.022} C_VEL
LIN {X 0,Y 159.569,Z 489.714,A -85,B 0,C 180,E1 -27590.654,E2 -27590.654} C_VEL
LIN {X 0,Y 164.531,Z 498.608,A -85,B 0,C 180,E1 -27595.294,E2 -27595.294} C_VEL
LIN {X 0,Y 170.629,Z 506.501,A -85,B 0,C 180,E1 -27599.876,E2 -27599.876} C_VEL
LIN {X 0,Y 177.783,Z 513.291,A -85,B 0,C 180,E1 -27604.225,E2 -27604.225} C_VEL
LIN {X 0,Y 184.748,Z 518.137,A -85,B 0,C 180,E1 -27607.642,E2 -27607.642} C_VEL
LIN {X 0,Y 193.102,Z 522.721,A -85,B 0,C 180,E1 -27611.13,E2 -27611.13} C_VEL
LIN {X 0,Y 203.877,Z 527.103,A -85,B 0,C 180,E1 -27614.837,E2 -27614.837} C_VEL
LIN {X 0,Y 217.473,Z 531.231,A -85,B 0,C 180,E1 -27618.82,E2 -27618.82} C_VEL
LIN {X 0,Y 227.385,Z 533.64,A -85,B 0,C 180,E1 -27621.507,E2 -27621.507} C_VEL
LIN {X 0,Y 233.549,Z 534.973,A -85,B 0,C 180,E1 -27623.229,E2 -27623.229} C_VEL
LIN {X 0,Y 239.792,Z 536.2,A -85,B 0,C 180,E1 -27625.189,E2 -27625.189} C_VEL
LIN {X 0,Y 243.487,Z 536.942,A -85,B 0,C 180,E1 -27626.691,E2 -27626.691} C_VEL
LIN {X 0,Y 246.813,Z 537.435,A -85,B 0,C 180,E1 -27628.368,E2 -27628.368} C_VEL
LIN {X 0,Y 248.647,Z 537.575,A -85,B 0,C 180,E1 -27630,E2 -27630} C_VEL
LIN {X 0,Y 246.802,Z 537.435,A -85,B 0,C 180,E1 -27631.632,E2 -27631.632} C_VEL
LIN {X 0,Y 243.48,Z 536.943,A -85,B 0,C 180,E1 -27633.309,E2 -27633.309} C_VEL
LIN {X 0,Y 239.051,Z 536.058,A -85,B 0,C 180,E1 -27635.06,E2 -27635.06} C_VEL
LIN {X 0,Y 233.051,Z 534.862,A -85,B 0,C 180,E1 -27636.928,E2 -27636.928} C_VEL
LIN {X 0,Y 225.624,Z 533.271,A -85,B 0,C 180,E1 -27638.96,E2 -27638.96} C_VEL
LIN {X 0,Y 215.363,Z 530.67,A -85,B 0,C 180,E1 -27641.769,E2 -27641.769} C_VEL
LIN {X 0,Y 200.344,Z 525.83,A -85,B 0,C 180,E1 -27646.298,E2 -27646.298} C_VEL
LIN {X 0,Y 188.055,Z 520.119,A -85,B 0,C 180,E1 -27650.889,E2 -27650.889} C_VEL
LIN {X 0,Y 178.746,Z 514.028,A -85,B 0,C 180,E1 -27655.271,E2 -27655.271} C_VEL
LIN {X 0,Y 171.731,Z 507.648,A -85,B 0,C 180,E1 -27659.412,E2 -27659.412} C_VEL
LIN {X 0,Y 165.662,Z 500.325,A -85,B 0,C 180,E1 -27663.751,E2 -27663.751} C_VEL
LIN {X 0,Y 161.262,Z 493.176,A -85,B 0,C 180,E1 -27667.598,E2 -27667.598} C_VEL
LIN {X 0,Y 157.473,Z 484.865,A -85,B 0,C 180,E1 -27671.624,E2 -27671.624} C_VEL
LIN {X 0,Y 154.694,Z 476.448,A -85,B 0,C 180,E1 -27675.238,E2 -27675.238} C_VEL
LIN {X 0,Y 152.218,Z 467.02,A -85,B 0,C 180,E1 -27678.859,E2 -27678.859} C_VEL
LIN {X 0,Y 150.295,Z 457.892,A -85,B 0,C 180,E1 -27681.941,E2 -27681.941} C_VEL
LIN {X 0,Y 148.504,Z 448.366,A -85,B 0,C 180,E1 -27684.777,E2 -27684.777} C_VEL
LIN {X 0,Y 146.407,Z 438.047,A -85,B 0,C 180,E1 -27687.622,E2 -27687.622} C_VEL
LIN {X 0,Y 144.004,Z 430.132,A -85,B 0,C 180,E1 -27690.087,E2 -27690.087} C_VEL
LIN {X 0,Y 140.706,Z 421.612,A -85,B 0,C 180,E1 -27693.476,E2 -27693.476} C_VEL
LIN {X 0,Y 137.594,Z 414.684,A -85,B 0,C 180,E1 -27697.13,E2 -27697.13} C_VEL
LIN {X 0,Y 134.468,Z 408.483,A -85,B 0,C 180,E1 -27701.577,E2 -27701.577} C_VEL
LIN {X 0,Y 132.443,Z 404.844,A -85,B 0,C 180,E1 -27705.206,E2 -27705.206} C_VEL
LIN {X 0,Y 130.822,Z 401.636,A -85,B 0,C 180,E1 -27709.135,E2 -27709.135} C_VEL
LIN {X 0,Y 129.175,Z 397.812,A -85,B 0,C 180,E1 -27717.078,E2 -27717.078} C_VEL
LIN {X 0,Y 129.11,Z 397.151,A -85,B 0,C 180,E1 -27720.002,E2 -27720.002} C_VEL
LIN {X 0,Y 129.18,Z 397.942,A -85,B 0,C 180,E1 -27722.73,E2 -27722.73} C_VEL
LIN {X 0,Y 131.084,Z 402.132,A -85,B 0,C 180,E1 -27731.209,E2 -27731.209} C_VEL
LIN {X 0,Y 133.307,Z 406.399,A -85,B 0,C 180,E1 -27736.07,E2 -27736.07} C_VEL
LIN {X 0,Y 135.239,Z 410.041,A -85,B 0,C 180,E1 -27739.25,E2 -27739.25} C_VEL
LIN {X 0,Y 137.614,Z 414.845,A -85,B 0,C 180,E1 -27742.527,E2 -27742.527} C_VEL
LIN {X 0,Y 139.541,Z 420.954,A -85,B 0,C 180,E1 -27745.078,E2 -27745.078} C_VEL
LIN {X 0,Y 140.839,Z 425.56,A -85,B 0,C 180,E1 -27746.688,E2 -27746.688} C_VEL
LIN {X 0,Y 138.72,Z 445.013,A -85,B 0,C 180,E1 -27747.465,E2 -27747.465} C_VEL
LIN {X 0,Y 135.719,Z 458.859,A -85,B 0,C 180,E1 -27748.322,E2 -27748.322} C_VEL
LIN {X 0,Y 132.429,Z 469.496,A -85,B 0,C 180,E1 -27749.271,E2 -27749.271} C_VEL
LIN {X 0,Y 128.461,Z 479.629,A -85,B 0,C 180,E1 -27750.498,E2 -27750.498} C_VEL
LIN {X 0,Y 124.198,Z 488.618,A -85,B 0,C 180,E1 -27751.92,E2 -27751.92} C_VEL
LIN {X 0,Y 119.376,Z 497.339,A -85,B 0,C 180,E1 -27753.741,E2 -27753.741} C_VEL
LIN {X 0,Y 114.667,Z 504.727,A -85,B 0,C 180,E1 -27755.7,E2 -27755.7} C_VEL
LIN {X 0,Y 109.5,Z 511.941,A -85,B 0,C 180,E1 -27758.167,E2 -27758.167} C_VEL
LIN {X 0,Y 104.577,Z 518.138,A -85,B 0,C 180,E1 -27760.885,E2 -27760.885} C_VEL
LIN {X 0,Y 98.797,Z 524.672,A -85,B 0,C 180,E1 -27764.656,E2 -27764.656} C_VEL
LIN {X 0,Y 94.62,Z 529.176,A -85,B 0,C 180,E1 -27768.051,E2 -27768.051} C_VEL
LIN {X 0,Y 88.936,Z 534.669,A -85,B 0,C 180,E1 -27773.654,E2 -27773.654} C_VEL
LIN {X 0,Y 84.147,Z 538.996,A -85,B 0,C 180,E1 -27779.927,E2 -27779.927} C_VEL
LIN {X 0,Y 81.512,Z 541.366,A -85,B 0,C 180,E1 -27784.463,E2 -27784.463} C_VEL
LIN {X 0,Y 79.521,Z 543.172,A -85,B 0,C 180,E1 -27789.298,E2 -27789.298} C_VEL
LIN {X 0,Y 77.134,Z 545.636,A -85,B 0,C 180,E1 -27799.501,E2 -27799.501} C_VEL
LIN {X 0,Y 76.734,Z 546.235,A -85,B 0,C 180,E1 -27804.745,E2 -27804.745} C_VEL
LIN {X 0,Y 76.781,Z 546.397,A -85,B 0,C 180,E1 -27810,E2 -27810} C_VEL
LIN {X 0,Y 76.71,Z 546.234,A -85,B 0,C 180,E1 -27815.257,E2 -27815.257} C_VEL
LIN {X 0,Y 77.118,Z 545.636,A -85,B 0,C 180,E1 -27820.501,E2 -27820.501} C_VEL
LIN {X 0,Y 79.521,Z 543.172,A -85,B 0,C 180,E1 -27830.702,E2 -27830.702} C_VEL
LIN {X 0,Y 82.771,Z 540.214,A -85,B 0,C 180,E1 -27837.839,E2 -27837.839} C_VEL
LIN {X 0,Y 87.206,Z 536.222,A -85,B 0,C 180,E1 -27844.341,E2 -27844.341} C_VEL
LIN {X 0,Y 92.702,Z 531.094,A -85,B 0,C 180,E1 -27850.12,E2 -27850.12} C_VEL
LIN {X 0,Y 97.769,Z 525.831,A -85,B 0,C 180,E1 -27854.494,E2 -27854.494} C_VEL
LIN {X 0,Y 103.374,Z 519.513,A -85,B 0,C 180,E1 -27858.403,E2 -27858.403} C_VEL
LIN {X 0,Y 108.254,Z 513.567,A -85,B 0,C 180,E1 -27861.173,E2 -27861.173} C_VEL
LIN {X 0,Y 113.367,Z 506.646,A -85,B 0,C 180,E1 -27863.697,E2 -27863.697} C_VEL
LIN {X 0,Y 118.684,Z 498.473,A -85,B 0,C 180,E1 -27865.997,E2 -27865.997} C_VEL
LIN {X 0,Y 123.505,Z 489.969,A -85,B 0,C 180,E1 -27867.826,E2 -27867.826} C_VEL
LIN {X 0,Y 127.726,Z 481.259,A -85,B 0,C 180,E1 -27869.287,E2 -27869.287} C_VEL
LIN {X 0,Y 131.723,Z 471.51,A -85,B 0,C 180,E1 -27870.496,E2 -27870.496} C_VEL
LIN {X 0,Y 134.96,Z 461.432,A -85,B 0,C 180,E1 -27871.49,E2 -27871.49} C_VEL
LIN {X 0,Y 137.424,Z 451.654,A -85,B 0,C 180,E1 -27872.16,E2 -27872.16} C_VEL
LIN {X 0,Y 139.108,Z 441.97,A -85,B 0,C 180,E1 -27872.676,E2 -27872.676} C_VEL
LIN {X 0,Y 140.845,Z 425.506,A -85,B 0,C 180,E1 -27873.313,E2 -27873.313} C_VEL
LIN {X 0,Y 138.388,Z 417.118,A -85,B 0,C 180,E1 -27876.431,E2 -27876.431} C_VEL
LIN {X 0,Y 137.006,Z 413.58,A -85,B 0,C 180,E1 -27878.262,E2 -27878.262} C_VEL
LIN {X 0,Y 134.49,Z 408.545,A -85,B 0,C 180,E1 -27881.923,E2 -27881.923} C_VEL
LIN {X 0,Y 132.534,Z 404.988,A -85,B 0,C 180,E1 -27885.409,E2 -27885.409} C_VEL
LIN {X 0,Y 130.813,Z 401.6,A -85,B 0,C 180,E1 -27889.551,E2 -27889.551} C_VEL
LIN {X 0,Y 129.137,Z 397.416,A -85,B 0,C 180,E1 -27898.439,E2 -27898.439} C_VEL
LIN {X 0,Y 129.104,Z 397.254,A -85,B 0,C 180,E1 -27900.778,E2 -27900.778} C_VEL
LIN {X 0,Y 129.182,Z 397.928,A -85,B 0,C 180,E1 -27903.117,E2 -27903.117} C_VEL
LIN {X 0,Y 130.821,Z 401.648,A -85,B 0,C 180,E1 -27910.866,E2 -27910.866} C_VEL
LIN {X 0,Y 133.21,Z 406.217,A -85,B 0,C 180,E1 -27916.275,E2 -27916.275} C_VEL
LIN {X 0,Y 135.197,Z 410,A -85,B 0,C 180,E1 -27919.578,E2 -27919.578} C_VEL
LIN {X 0,Y 137.903,Z 415.355,A -85,B 0,C 180,E1 -27923.262,E2 -27923.262} C_VEL
LIN {X 0,Y 140.941,Z 422.221,A -85,B 0,C 180,E1 -27926.785,E2 -27926.785} C_VEL
LIN {X 0,Y 141.98,Z 424.784,A -85,B 0,C 180,E1 -27927.884,E2 -27927.884} C_VEL
LIN {X 0,Y 142.9,Z 427.713,A -85,B 0,C 180,E1 -27928.872,E2 -27928.872} C_VEL
LIN {X 0,Y 143.763,Z 432.831,A -85,B 0,C 180,E1 -27930.017,E2 -27930.017} C_VEL
LIN {X 0,Y 144.118,Z 445.899,A -85,B 0,C 180,E1 -27932.135,E2 -27932.135} C_VEL
LIN {X 0,Y 144.295,Z 451.236,A -85,B 0,C 180,E1 -27933.267,E2 -27933.267} C_VEL
LIN {X 0,Y 144.452,Z 452.882,A -85,B 0,C 180,E1 -27933.725,E2 -27933.725} C_VEL
LIN {X 0,Y 146.124,Z 464.501,A -85,B 0,C 180,E1 -27937.539,E2 -27937.539} C_VEL
LIN {X 0,Y 147.728,Z 473.259,A -85,B 0,C 180,E1 -27940.853,E2 -27940.853} C_VEL
LIN {X 0,Y 149.828,Z 482.331,A -85,B 0,C 180,E1 -27944.715,E2 -27944.715} C_VEL
LIN {X 0,Y 152.693,Z 491.125,A -85,B 0,C 180,E1 -27948.966,E2 -27948.966} C_VEL
LIN {X 0,Y 156.431,Z 498.896,A -85,B 0,C 180,E1 -27953.223,E2 -27953.223} C_VEL
LIN {X 0,Y 161.29,Z 506.2,A -85,B 0,C 180,E1 -27957.657,E2 -27957.657} C_VEL
LIN {X 0,Y 167.184,Z 512.658,A -85,B 0,C 180,E1 -27961.978,E2 -27961.978} C_VEL
LIN {X 0,Y 174.393,Z 518.438,A -85,B 0,C 180,E1 -27966.235,E2 -27966.235} C_VEL
LIN {X 0,Y 181.41,Z 522.628,A -85,B 0,C 180,E1 -27969.595,E2 -27969.595} C_VEL
LIN {X 0,Y 190.742,Z 526.826,A -85,B 0,C 180,E1 -27973.328,E2 -27973.328} C_VEL
LIN {X 0,Y 205.772,Z 531.55,A -85,B 0,C 180,E1 -27978.175,E2 -27978.175} C_VEL
LIN {X 0,Y 214.308,Z 533.584,A -85,B 0,C 180,E1 -27980.563,E2 -27980.563} C_VEL
LIN {X 0,Y 222.386,Z 535.157,A -85,B 0,C 180,E1 -27982.738,E2 -27982.738} C_VEL
LIN {X 0,Y 229.364,Z 536.321,A -85,B 0,C 180,E1 -27984.726,E2 -27984.726} C_VEL
LIN {X 0,Y 232.572,Z 536.834,A -85,B 0,C 180,E1 -27985.707,E2 -27985.707} C_VEL
LIN {X 0,Y 234.951,Z 537.177,A -85,B 0,C 180,E1 -27986.57,E2 -27986.57} C_VEL
LIN {X 0,Y 239.045,Z 537.66,A -85,B 0,C 180,E1 -27988.36,E2 -27988.36} C_VEL
LIN {X 0,Y 241.292,Z 537.772,A -85,B 0,C 180,E1 -27990,E2 -27990} C_VEL
LIN {X 0,Y 238.924,Z 537.65,A -85,B 0,C 180,E1 -27991.686,E2 -27991.686} C_VEL
LIN {X 0,Y 234.951,Z 537.178,A -85,B 0,C 180,E1 -27993.43,E2 -27993.43} C_VEL
LIN {X 0,Y 232.573,Z 536.832,A -85,B 0,C 180,E1 -27994.295,E2 -27994.295} C_VEL
LIN {X 0,Y 226.216,Z 535.837,A -85,B 0,C 180,E1 -27996.203,E2 -27996.203} C_VEL
LIN {X 0,Y 219.955,Z 534.697,A -85,B 0,C 180,E1 -27997.907,E2 -27997.907} C_VEL
LIN {X 0,Y 207.794,Z 532.055,A -85,B 0,C 180,E1 -28001.242,E2 -28001.242} C_VEL
LIN {X 0,Y 196.224,Z 528.761,A -85,B 0,C 180,E1 -28004.757,E2 -28004.757} C_VEL
LIN {X 0,Y 185.458,Z 524.578,A -85,B 0,C 180,E1 -28008.673,E2 -28008.673} C_VEL
LIN {X 0,Y 175.708,Z 519.291,A -85,B 0,C 180,E1 -28013.084,E2 -28013.084} C_VEL
LIN {X 0,Y 168.161,Z 513.578,A -85,B 0,C 180,E1 -28017.369,E2 -28017.369} C_VEL
LIN {X 0,Y 162.663,Z 507.927,A -85,B 0,C 180,E1 -28021.229,E2 -28021.229} C_VEL
LIN {X 0,Y 157.791,Z 501.304,A -85,B 0,C 180,E1 -28025.381,E2 -28025.381} C_VEL
LIN {X 0,Y 154.192,Z 494.574,A -85,B 0,C 180,E1 -28029.211,E2 -28029.211} C_VEL
LIN {X 0,Y 151.307,Z 487.262,A -85,B 0,C 180,E1 -28032.986,E2 -28032.986} C_VEL
LIN {X 0,Y 148.475,Z 477.067,A -85,B 0,C 180,E1 -28037.596,E2 -28037.596} C_VEL
LIN {X 0,Y 146.793,Z 468.505,A -85,B 0,C 180,E1 -28040.999,E2 -28040.999} C_VEL
LIN {X 0,Y 145.22,Z 458.454,A -85,B 0,C 180,E1 -28044.499,E2 -28044.499} C_VEL
LIN {X 0,Y 143.839,Z 448.653,A -85,B 0,C 180,E1 -28047.491,E2 -28047.491} C_VEL
LIN {X 0,Y 142.167,Z 439.333,A -85,B 0,C 180,E1 -28050.273,E2 -28050.273} C_VEL
LIN {X 0,Y 139.732,Z 431.269,A -85,B 0,C 180,E1 -28053.188,E2 -28053.188} C_VEL
LIN {X 0,Y 136.772,Z 423.666,A -85,B 0,C 180,E1 -28056.76,E2 -28056.76} C_VEL
LIN {X 0,Y 134.185,Z 417.771,A -85,B 0,C 180,E1 -28060.422,E2 -28060.422} C_VEL
LIN {X 0,Y 132.1,Z 413.585,A -85,B 0,C 180,E1 -28063.981,E2 -28063.981} C_VEL
LIN {X 0,Y 130.934,Z 411.274,A -85,B 0,C 180,E1 -28066.419,E2 -28066.419} C_VEL
LIN {X 0,Y 129.665,Z 408.477,A -85,B 0,C 180,E1 -28069.868,E2 -28069.868} C_VEL
LIN {X 0,Y 128.251,Z 404.44,A -85,B 0,C 180,E1 -28078.432,E2 -28078.432} C_VEL
LIN {X 0,Y 128.246,Z 404.335,A -85,B 0,C 180,E1 -28080.787,E2 -28080.787} C_VEL
LIN {X 0,Y 129.884,Z 408.954,A -85,B 0,C 180,E1 -28090.426,E2 -28090.426} C_VEL
LIN {X 0,Y 131.812,Z 412.986,A -85,B 0,C 180,E1 -28095.067,E2 -28095.067} C_VEL
LIN {X 0,Y 133.503,Z 416.409,A -85,B 0,C 180,E1 -28098.117,E2 -28098.117} C_VEL
LIN {X 0,Y 135.506,Z 420.93,A -85,B 0,C 180,E1 -28101.177,E2 -28101.177} C_VEL
LIN {X 0,Y 137.218,Z 427.079,A -85,B 0,C 180,E1 -28103.725,E2 -28103.725} C_VEL
LIN {X 0,Y 137.504,Z 428.233,A -85,B 0,C 180,E1 -28104.137,E2 -28104.137} C_VEL
LIN {X 0,Y 135.372,Z 446.237,A -85,B 0,C 180,E1 -28104.871,E2 -28104.871} C_VEL
LIN {X 0,Y 132.504,Z 458.665,A -85,B 0,C 180,E1 -28105.623,E2 -28105.623} C_VEL
LIN {X 0,Y 129.111,Z 469.302,A -85,B 0,C 180,E1 -28106.526,E2 -28106.526} C_VEL
LIN {X 0,Y 125.01,Z 479.436,A -85,B 0,C 180,E1 -28107.695,E2 -28107.695} C_VEL
LIN {X 0,Y 120.593,Z 488.424,A -85,B 0,C 180,E1 -28109.055,E2 -28109.055} C_VEL
LIN {X 0,Y 115.588,Z 497.146,A -85,B 0,C 180,E1 -28110.817,E2 -28110.817} C_VEL
LIN {X 0,Y 110.671,Z 504.533,A -85,B 0,C 180,E1 -28112.712,E2 -28112.712} C_VEL
LIN {X 0,Y 105.246,Z 511.746,A -85,B 0,C 180,E1 -28115.115,E2 -28115.115} C_VEL
LIN {X 0,Y 100.055,Z 517.944,A -85,B 0,C 180,E1 -28117.796,E2 -28117.796} C_VEL
LIN {X 0,Y 93.926,Z 524.477,A -85,B 0,C 180,E1 -28121.563,E2 -28121.563} C_VEL
LIN {X 0,Y 88.216,Z 530.074,A -85,B 0,C 180,E1 -28126.031,E2 -28126.031} C_VEL
LIN {X 0,Y 83.311,Z 534.474,A -85,B 0,C 180,E1 -28130.753,E2 -28130.753} C_VEL
LIN {X 0,Y 78.061,Z 538.801,A -85,B 0,C 180,E1 -28137.304,E2 -28137.304} C_VEL
LIN {X 0,Y 75.139,Z 541.171,A -85,B 0,C 180,E1 -28142.118,E2 -28142.118} C_VEL
LIN {X 0,Y 72.893,Z 542.977,A -85,B 0,C 180,E1 -28147.316,E2 -28147.316} C_VEL
LIN {X 0,Y 70.153,Z 545.442,A -85,B 0,C 180,E1 -28158.442,E2 -28158.442} C_VEL
LIN {X 0,Y 69.646,Z 546.04,A -85,B 0,C 180,E1 -28164.209,E2 -28164.209} C_VEL
LIN {X 0,Y 69.701,Z 546.204,A -85,B 0,C 180,E1 -28170,E2 -28170} C_VEL
LIN {X 0,Y 69.622,Z 546.04,A -85,B 0,C 180,E1 -28175.793,E2 -28175.793} C_VEL
LIN {X 0,Y 70.118,Z 545.441,A -85,B 0,C 180,E1 -28181.564,E2 -28181.564} C_VEL
LIN {X 0,Y 72.893,Z 542.977,A -85,B 0,C 180,E1 -28192.684,E2 -28192.684} C_VEL
LIN {X 0,Y 76.545,Z 540.02,A -85,B 0,C 180,E1 -28200.33,E2 -28200.33} C_VEL
LIN {X 0,Y 81.413,Z 536.028,A -85,B 0,C 180,E1 -28207.176,E2 -28207.176} C_VEL
LIN {X 0,Y 87.366,Z 530.899,A -85,B 0,C 180,E1 -28213.138,E2 -28213.138} C_VEL
LIN {X 0,Y 92.813,Z 525.636,A -85,B 0,C 180,E1 -28217.583,E2 -28217.583} C_VEL
LIN {X 0,Y 98.795,Z 519.319,A -85,B 0,C 180,E1 -28221.489,E2 -28221.489} C_VEL
LIN {X 0,Y 103.939,Z 513.372,A -85,B 0,C 180,E1 -28224.231,E2 -28224.231} C_VEL
LIN {X 0,Y 109.299,Z 506.451,A -85,B 0,C 180,E1 -28226.708,E2 -28226.708} C_VEL
LIN {X 0,Y 114.866,Z 498.279,A -85,B 0,C 180,E1 -28228.932,E2 -28228.932} C_VEL
LIN {X 0,Y 119.879,Z 489.775,A -85,B 0,C 180,E1 -28230.696,E2 -28230.696} C_VEL
LIN {X 0,Y 124.256,Z 481.065,A -85,B 0,C 180,E1 -28232.097,E2 -28232.097} C_VEL
LIN {X 0,Y 128.379,Z 471.316,A -85,B 0,C 180,E1 -28233.252,E2 -28233.252} C_VEL
LIN {X 0,Y 131.727,Z 461.238,A -85,B 0,C 180,E1 -28234.198,E2 -28234.198} C_VEL
LIN {X 0,Y 134.291,Z 451.306,A -85,B 0,C 180,E1 -28234.846,E2 -28234.846} C_VEL
LIN {X 0,Y 136.057,Z 441.287,A -85,B 0,C 180,E1 -28235.359,E2 -28235.359} C_VEL
LIN {X 0,Y 137.505,Z 428.222,A -85,B 0,C 180,E1 -28235.863,E2 -28235.863} C_VEL
LIN {X 0,Y 135.575,Z 421.112,A -85,B 0,C 180,E1 -28238.722,E2 -28238.722} C_VEL
LIN {X 0,Y 133.771,Z 416.951,A -85,B 0,C 180,E1 -28241.45,E2 -28241.45} C_VEL
LIN {X 0,Y 131.462,Z 412.141,A -85,B 0,C 180,E1 -28245.683,E2 -28245.683} C_VEL
LIN {X 0,Y 129.739,Z 408.516,A -85,B 0,C 180,E1 -28250.055,E2 -28250.055} C_VEL
LIN {X 0,Y 128.246,Z 404.335,A -85,B 0,C 180,E1 -28259.213,E2 -28259.213} C_VEL
LIN {X 0,Y 128.264,Z 404.534,A -85,B 0,C 180,E1 -28261.961,E2 -28261.961} C_VEL
LIN {X 0,Y 129.927,Z 409.064,A -85,B 0,C 180,E1 -28270.941,E2 -28270.941} C_VEL
LIN {X 0,Y 131.772,Z 412.877,A -85,B 0,C 180,E1 -28275.365,E2 -28275.365} C_VEL
LIN {X 0,Y 133.558,Z 416.531,A -85,B 0,C 180,E1 -28278.593,E2 -28278.593} C_VEL
LIN {X 0,Y 136.167,Z 422.246,A -85,B 0,C 180,E1 -28282.441,E2 -28282.441} C_VEL
LIN {X 0,Y 138.689,Z 428.491,A -85,B 0,C 180,E1 -28285.613,E2 -28285.613} C_VEL
LIN {X 0,Y 141.225,Z 436.041,A -85,B 0,C 180,E1 -28288.617,E2 -28288.617} C_VEL
LIN {X 0,Y 143.288,Z 444.772,A -85,B 0,C 180,E1 -28291.407,E2 -28291.407} C_VEL
LIN {X 0,Y 144.452,Z 452.882,A -85,B 0,C 180,E1 -28293.725,E2 -28293.725} C_VEL
LIN {X 0,Y 144.688,Z 457.807,A -85,B 0,C 180,E1 -28295.025,E2 -28295.025} C_VEL
LIN {X 0,Y 143.898,Z 466.455,A -85,B 0,C 180,E1 -28296.919,E2 -28296.919} C_VEL
LIN {X 0,Y 142.897,Z 474.76,A -85,B 0,C 180,E1 -28298.995,E2 -28298.995} C_VEL
LIN {X 0,Y 142.941,Z 479.148,A -85,B 0,C 180,E1 -28300.546,E2 -28300.546} C_VEL
LIN {X 0,Y 145.234,Z 489.534,A -85,B 0,C 180,E1 -28305.54,E2 -28305.54} C_VEL
LIN {X 0,Y 148.157,Z 498.075,A -85,B 0,C 180,E1 -28310.273,E2 -28310.273} C_VEL
LIN {X 0,Y 152.202,Z 505.66,A -85,B 0,C 180,E1 -28315.043,E2 -28315.043} C_VEL
LIN {X 0,Y 157.65,Z 512.631,A -85,B 0,C 180,E1 -28319.943,E2 -28319.943} C_VEL
LIN {X 0,Y 164.45,Z 518.73,A -85,B 0,C 180,E1 -28324.7,E2 -28324.7} C_VEL
LIN {X 0,Y 172.835,Z 523.971,A -85,B 0,C 180,E1 -28329.264,E2 -28329.264} C_VEL
LIN {X 0,Y 183.084,Z 528.477,A -85,B 0,C 180,E1 -28333.667,E2 -28333.667} C_VEL
LIN {X 0,Y 194.321,Z 531.956,A -85,B 0,C 180,E1 -28337.55,E2 -28337.55} C_VEL
LIN {X 0,Y 206.318,Z 534.61,A -85,B 0,C 180,E1 -28341.053,E2 -28341.053} C_VEL
LIN {X 0,Y 218.898,Z 536.575,A -85,B 0,C 180,E1 -28344.426,E2 -28344.426} C_VEL
LIN {X 0,Y 225.812,Z 537.429,A -85,B 0,C 180,E1 -28346.431,E2 -28346.431} C_VEL
LIN {X 0,Y 231.968,Z 537.95,A -85,B 0,C 180,E1 -28348.823,E2 -28348.823} C_VEL
LIN {X 0,Y 233.812,Z 537.972,A -85,B 0,C 180,E1 -28350,E2 -28350} C_VEL
LIN {X 0,Y 231.968,Z 537.95,A -85,B 0,C 180,E1 -28351.168,E2 -28351.168} C_VEL
LIN {X 0,Y 225.829,Z 537.429,A -85,B 0,C 180,E1 -28353.568,E2 -28353.568} C_VEL
LIN {X 0,Y 218.898,Z 536.575,A -85,B 0,C 180,E1 -28355.574,E2 -28355.574} C_VEL
LIN {X 0,Y 206.318,Z 534.61,A -85,B 0,C 180,E1 -28358.947,E2 -28358.947} C_VEL
LIN {X 0,Y 194.026,Z 531.872,A -85,B 0,C 180,E1 -28362.552,E2 -28362.552} C_VEL
LIN {X 0,Y 180.42,Z 527.505,A -85,B 0,C 180,E1 -28367.385,E2 -28367.385} C_VEL
LIN {X 0,Y 168.148,Z 521.305,A -85,B 0,C 180,E1 -28373.148,E2 -28373.148} C_VEL
LIN {X 0,Y 159.822,Z 514.773,A -85,B 0,C 180,E1 -28378.424,E2 -28378.424} C_VEL
LIN {X 0,Y 154.517,Z 508.934,A -85,B 0,C 180,E1 -28382.712,E2 -28382.712} C_VEL
LIN {X 0,Y 149.782,Z 501.571,A -85,B 0,C 180,E1 -28387.587,E2 -28387.587} C_VEL
LIN {X 0,Y 146.389,Z 493.7,A -85,B 0,C 180,E1 -28392.23,E2 -28392.23} C_VEL
LIN {X 0,Y 144.35,Z 486.325,A -85,B 0,C 180,E1 -28396.071,E2 -28396.071} C_VEL
LIN {X 0,Y 142.949,Z 479.141,A -85,B 0,C 180,E1 -28399.452,E2 -28399.452} C_VEL
LIN {X 0,Y 141.567,Z 469.574,A -85,B 0,C 180,E1 -28403.437,E2 -28403.437} C_VEL
LIN {X 0,Y 140.5,Z 459.361,A -85,B 0,C 180,E1 -28407.118,E2 -28407.118} C_VEL
LIN {X 0,Y 139.483,Z 448.615,A -85,B 0,C 180,E1 -28410.474,E2 -28410.474} C_VEL
LIN {X 0,Y 138.138,Z 440.695,A -85,B 0,C 180,E1 -28413.16,E2 -28413.16} C_VEL
LIN {X 0,Y 135.84,Z 432.883,A -85,B 0,C 180,E1 -28416.465,E2 -28416.465} C_VEL
LIN {X 0,Y 133.42,Z 426.468,A -85,B 0,C 180,E1 -28419.979,E2 -28419.979} C_VEL
LIN {X 0,Y 131.096,Z 421.071,A -85,B 0,C 180,E1 -28424.055,E2 -28424.055} C_VEL
LIN {X 0,Y 129.493,Z 417.647,A -85,B 0,C 180,E1 -28427.66,E2 -28427.66} C_VEL
LIN {X 0,Y 128.548,Z 415.324,A -85,B 0,C 180,E1 -28430.562,E2 -28430.562} C_VEL
LIN {X 0,Y 127.37,Z 411.374,A -85,B 0,C 180,E1 -28439.211,E2 -28439.211} C_VEL
LIN {X 0,Y 127.376,Z 411.574,A -85,B 0,C 180,E1 -28441.187,E2 -28441.187} C_VEL
LIN {X 0,Y 128.715,Z 415.724,A -85,B 0,C 180,E1 -28449.628,E2 -28449.628} C_VEL
LIN {X 0,Y 130.364,Z 419.521,A -85,B 0,C 180,E1 -28454.04,E2 -28454.04} C_VEL
LIN {X 0,Y 131.873,Z 422.891,A -85,B 0,C 180,E1 -28457.046,E2 -28457.046} C_VEL
LIN {X 0,Y 133.414,Z 426.762,A -85,B 0,C 180,E1 -28459.674,E2 -28459.674} C_VEL
LIN {X 0,Y 134.442,Z 431.021,A -85,B 0,C 180,E1 -28461.466,E2 -28461.466} C_VEL
LIN {X 0,Y 132.443,Z 446.551,A -85,B 0,C 180,E1 -28462.113,E2 -28462.113} C_VEL
LIN {X 0,Y 129.593,Z 458.472,A -85,B 0,C 180,E1 -28462.793,E2 -28462.793} C_VEL
LIN {X 0,Y 126.465,Z 468.219,A -85,B 0,C 180,E1 -28463.577,E2 -28463.577} C_VEL
LIN {X 0,Y 121.873,Z 479.242,A -85,B 0,C 180,E1 -28464.739,E2 -28464.739} C_VEL
LIN {X 0,Y 117.307,Z 488.23,A -85,B 0,C 180,E1 -28466.019,E2 -28466.019} C_VEL
LIN {X 0,Y 112.115,Z 496.952,A -85,B 0,C 180,E1 -28467.697,E2 -28467.697} C_VEL
LIN {X 0,Y 106.999,Z 504.339,A -85,B 0,C 180,E1 -28469.51,E2 -28469.51} C_VEL
LIN {X 0,Y 101.318,Z 511.552,A -85,B 0,C 180,E1 -28471.82,E2 -28471.82} C_VEL
LIN {X 0,Y 95.863,Z 517.749,A -85,B 0,C 180,E1 -28474.436,E2 -28474.436} C_VEL
LIN {X 0,Y 89.355,Z 524.283,A -85,B 0,C 180,E1 -28478.14,E2 -28478.14} C_VEL
LIN {X 0,Y 83.861,Z 529.349,A -85,B 0,C 180,E1 -28482.105,E2 -28482.105} C_VEL
LIN {X 0,Y 77.933,Z 534.28,A -85,B 0,C 180,E1 -28487.442,E2 -28487.442} C_VEL
LIN {X 0,Y 72.169,Z 538.607,A -85,B 0,C 180,E1 -28494.248,E2 -28494.248} C_VEL
LIN {X 0,Y 68.921,Z 540.976,A -85,B 0,C 180,E1 -28499.346,E2 -28499.346} C_VEL
LIN {X 0,Y 64.456,Z 544.179,A -85,B 0,C 180,E1 -28510.907,E2 -28510.907} C_VEL
LIN {X 0,Y 63.187,Z 545.247,A -85,B 0,C 180,E1 -28517.147,E2 -28517.147} C_VEL
LIN {X 0,Y 62.576,Z 545.846,A -85,B 0,C 180,E1 -28523.552,E2 -28523.552} C_VEL
LIN {X 0,Y 62.61,Z 546.01,A -85,B 0,C 180,E1 -28530,E2 -28530} C_VEL
LIN {X 0,Y 62.556,Z 545.845,A -85,B 0,C 180,E1 -28536.451,E2 -28536.451} C_VEL
LIN {X 0,Y 63.159,Z 545.246,A -85,B 0,C 180,E1 -28542.858,E2 -28542.858} C_VEL
LIN {X 0,Y 66.354,Z 542.782,A -85,B 0,C 180,E1 -28555.066,E2 -28555.066} C_VEL
LIN {X 0,Y 70.492,Z 539.825,A -85,B 0,C 180,E1 -28563.253,E2 -28563.253} C_VEL
LIN {X 0,Y 75.857,Z 535.833,A -85,B 0,C 180,E1 -28570.43,E2 -28570.43} C_VEL
LIN {X 0,Y 81.527,Z 531.374,A -85,B 0,C 180,E1 -28575.862,E2 -28575.862} C_VEL
LIN {X 0,Y 88.157,Z 525.44,A -85,B 0,C 180,E1 -28581.011,E2 -28581.011} C_VEL
LIN {X 0,Y 94.533,Z 519.125,A -85,B 0,C 180,E1 -28584.862,E2 -28584.862} C_VEL
LIN {X 0,Y 99.941,Z 513.178,A -85,B 0,C 180,E1 -28587.547,E2 -28587.547} C_VEL
LIN {X 0,Y 105.559,Z 506.257,A -85,B 0,C 180,E1 -28589.941,E2 -28589.941} C_VEL
LIN {X 0,Y 111.372,Z 498.085,A -85,B 0,C 180,E1 -28592.06,E2 -28592.06} C_VEL
LIN {X 0,Y 116.568,Z 489.581,A -85,B 0,C 180,E1 -28593.741,E2 -28593.741} C_VEL
LIN {X 0,Y 121.102,Z 480.872,A -85,B 0,C 180,E1 -28595.06,E2 -28595.06} C_VEL
LIN {X 0,Y 124.908,Z 472.185,A -85,B 0,C 180,E1 -28596.077,E2 -28596.077} C_VEL
LIN {X 0,Y 128.54,Z 461.898,A -85,B 0,C 180,E1 -28596.979,E2 -28596.979} C_VEL
LIN {X 0,Y 131.292,Z 451.738,A -85,B 0,C 180,E1 -28597.615,E2 -28597.615} C_VEL
LIN {X 0,Y 133.153,Z 441.831,A -85,B 0,C 180,E1 -28598.102,E2 -28598.102} C_VEL
LIN {X 0,Y 134.442,Z 431.022,A -85,B 0,C 180,E1 -28598.534,E2 -28598.534} C_VEL
LIN {X 0,Y 133.098,Z 425.732,A -85,B 0,C 180,E1 -28600.869,E2 -28600.869} C_VEL
LIN {X 0,Y 130.996,Z 420.864,A -85,B 0,C 180,E1 -28604.637,E2 -28604.637} C_VEL
LIN {X 0,Y 129.488,Z 417.64,A -85,B 0,C 180,E1 -28608.056,E2 -28608.056} C_VEL
LIN {X 0,Y 128.425,Z 415.178,A -85,B 0,C 180,E1 -28611.343,E2 -28611.343} C_VEL
LIN {X 0,Y 127.375,Z 411.371,A -85,B 0,C 180,E1 -28619.405,E2 -28619.405} C_VEL
LIN {X 0,Y 127.371,Z 411.707,A -85,B 0,C 180,E1 -28621.777,E2 -28621.777} C_VEL
LIN {X 0,Y 128.715,Z 415.756,A -85,B 0,C 180,E1 -28630.022,E2 -28630.022} C_VEL
LIN {X 0,Y 130.412,Z 419.632,A -85,B 0,C 180,E1 -28634.531,E2 -28634.531} C_VEL
LIN {X 0,Y 132.141,Z 423.48,A -85,B 0,C 180,E1 -28637.905,E2 -28637.905} C_VEL
LIN {X 0,Y 134.437,Z 429.057,A -85,B 0,C 180,E1 -28641.564,E2 -28641.564} C_VEL
LIN {X 0,Y 136.929,Z 436.461,A -85,B 0,C 180,E1 -28645.151,E2 -28645.151} C_VEL
LIN {X 0,Y 138.777,Z 443.777,A -85,B 0,C 180,E1 -28647.931,E2 -28647.931} C_VEL
LIN {X 0,Y 139.902,Z 451.965,A -85,B 0,C 180,E1 -28650.529,E2 -28650.529} C_VEL
LIN {X 0,Y 140.934,Z 463.399,A -85,B 0,C 180,E1 -28654.272,E2 -28654.272} C_VEL
LIN {X 0,Y 142.064,Z 473.666,A -85,B 0,C 180,E1 -28658.194,E2 -28658.194} C_VEL
LIN {X 0,Y 142.941,Z 479.148,A -85,B 0,C 180,E1 -28660.546,E2 -28660.546} C_VEL
LIN {X 0,Y 143.137,Z 483.419,A -85,B 0,C 180,E1 -28662.198,E2 -28662.198} C_VEL
LIN {X 0,Y 142.07,Z 490.868,A -85,B 0,C 180,E1 -28664.826,E2 -28664.826} C_VEL
LIN {X 0,Y 141.262,Z 497.84,A -85,B 0,C 180,E1 -28667.658,E2 -28667.658} C_VEL
LIN {X 0,Y 141.888,Z 501.138,A -85,B 0,C 180,E1 -28669.564,E2 -28669.564} C_VEL
LIN {X 0,Y 144.622,Z 506.762,A -85,B 0,C 180,E1 -28673.381,E2 -28673.381} C_VEL
LIN {X 0,Y 148.987,Z 513.093,A -85,B 0,C 180,E1 -28678.11,E2 -28678.11} C_VEL
LIN {X 0,Y 154.86,Z 519.015,A -85,B 0,C 180,E1 -28683.011,E2 -28683.011} C_VEL
LIN {X 0,Y 162.831,Z 524.522,A -85,B 0,C 180,E1 -28688.113,E2 -28688.113} C_VEL
LIN {X 0,Y 170.171,Z 528.099,A -85,B 0,C 180,E1 -28691.78,E2 -28691.78} C_VEL
LIN {X 0,Y 182.368,Z 532.192,A -85,B 0,C 180,E1 -28696.631,E2 -28696.631} C_VEL
LIN {X 0,Y 192.704,Z 534.594,A -85,B 0,C 180,E1 -28699.957,E2 -28699.957} C_VEL
LIN {X 0,Y 205.154,Z 536.578,A -85,B 0,C 180,E1 -28703.433,E2 -28703.433} C_VEL
LIN {X 0,Y 215.66,Z 537.709,A -85,B 0,C 180,E1 -28706.263,E2 -28706.263} C_VEL
LIN {X 0,Y 221.897,Z 538.113,A -85,B 0,C 180,E1 -28708.185,E2 -28708.185} C_VEL
LIN {X 0,Y 224.908,Z 538.192,A -85,B 0,C 180,E1 -28709.31,E2 -28709.31} C_VEL
LIN {X 0,Y 226.169,Z 538.177,A -85,B 0,C 180,E1 -28710,E2 -28710} C_VEL
LIN {X 0,Y 224.908,Z 538.193,A -85,B 0,C 180,E1 -28710.685,E2 -28710.685} C_VEL
LIN {X 0,Y 221.903,Z 538.112,A -85,B 0,C 180,E1 -28711.815,E2 -28711.815} C_VEL
LIN {X 0,Y 215.667,Z 537.709,A -85,B 0,C 180,E1 -28713.737,E2 -28713.737} C_VEL
LIN {X 0,Y 205.148,Z 536.586,A -85,B 0,C 180,E1 -28716.554,E2 -28716.554} C_VEL
LIN {X 0,Y 190.781,Z 534.237,A -85,B 0,C 180,E1 -28720.614,E2 -28720.614} C_VEL
LIN {X 0,Y 175.436,Z 530.084,A -85,B 0,C 180,E1 -28725.967,E2 -28725.967} C_VEL
LIN {X 0,Y 165.198,Z 525.791,A -85,B 0,C 180,E1 -28730.623,E2 -28730.623} C_VEL
LIN {X 0,Y 158.379,Z 521.792,A -85,B 0,C 180,E1 -28734.543,E2 -28734.543} C_VEL
LIN {X 0,Y 150.647,Z 515.029,A -85,B 0,C 180,E1 -28740.344,E2 -28740.344} C_VEL
LIN {X 0,Y 145.894,Z 509.003,A -85,B 0,C 180,E1 -28745.026,E2 -28745.026} C_VEL
LIN {X 0,Y 142.161,Z 501.838,A -85,B 0,C 180,E1 -28749.991,E2 -28749.991} C_VEL
LIN {X 0,Y 139.83,Z 494.952,A -85,B 0,C 180,E1 -28754.261,E2 -28754.261} C_VEL
LIN {X 0,Y 138.188,Z 486.998,A -85,B 0,C 180,E1 -28758.614,E2 -28758.614} C_VEL
LIN {X 0,Y 137.108,Z 477.882,A -85,B 0,C 180,E1 -28762.969,E2 -28762.969} C_VEL
LIN {X 0,Y 136.538,Z 469.319,A -85,B 0,C 180,E1 -28766.553,E2 -28766.553} C_VEL
LIN {X 0,Y 136.093,Z 459.289,A -85,B 0,C 180,E1 -28770.198,E2 -28770.198} C_VEL
LIN {X 0,Y 135.568,Z 450.121,A -85,B 0,C 180,E1 -28773.235,E2 -28773.235} C_VEL
LIN {X 0,Y 134.636,Z 443.532,A -85,B 0,C 180,E1 -28775.729,E2 -28775.729} C_VEL
LIN {X 0,Y 132.65,Z 435.89,A -85,B 0,C 180,E1 -28779.352,E2 -28779.352} C_VEL
LIN {X 0,Y 130.541,Z 429.941,A -85,B 0,C 180,E1 -28783.181,E2 -28783.181} C_VEL
LIN {X 0,Y 128.814,Z 425.682,A -85,B 0,C 180,E1 -28786.996,E2 -28786.996} C_VEL
LIN {X 0,Y 127.366,Z 422.044,A -85,B 0,C 180,E1 -28791.574,E2 -28791.574} C_VEL
LIN {X 0,Y 126.504,Z 418.379,A -85,B 0,C 180,E1 -28799.61,E2 -28799.61} C_VEL
LIN {X 0,Y 126.49,Z 418.722,A -85,B 0,C 180,E1 -28801.034,E2 -28801.034} C_VEL
LIN {X 0,Y 127.591,Z 422.615,A -85,B 0,C 180,E1 -28808.914,E2 -28808.914} C_VEL
LIN {X 0,Y 128.995,Z 426.165,A -85,B 0,C 180,E1 -28813.085,E2 -28813.085} C_VEL
LIN {X 0,Y 130.534,Z 429.929,A -85,B 0,C 180,E1 -28816.421,E2 -28816.421} C_VEL
LIN {X 0,Y 131.453,Z 432.794,A -85,B 0,C 180,E1 -28818.207,E2 -28818.207} C_VEL
LIN {X 0,Y 131.677,Z 433.885,A -85,B 0,C 180,E1 -28818.679,E2 -28818.679} C_VEL
LIN {X 0,Y 129.64,Z 447.607,A -85,B 0,C 180,E1 -28819.255,E2 -28819.255} C_VEL
LIN {X 0,Y 127.016,Z 458.278,A -85,B 0,C 180,E1 -28819.846,E2 -28819.846} C_VEL
LIN {X 0,Y 123.612,Z 468.488,A -85,B 0,C 180,E1 -28820.603,E2 -28820.603} C_VEL
LIN {X 0,Y 119.078,Z 479.048,A -85,B 0,C 180,E1 -28821.637,E2 -28821.637} C_VEL
LIN {X 0,Y 114.37,Z 488.036,A -85,B 0,C 180,E1 -28822.82,E2 -28822.82} C_VEL
LIN {X 0,Y 108.986,Z 496.757,A -85,B 0,C 180,E1 -28824.379,E2 -28824.379} C_VEL
LIN {X 0,Y 103.674,Z 504.145,A -85,B 0,C 180,E1 -28826.079,E2 -28826.079} C_VEL
LIN {X 0,Y 97.748,Z 511.357,A -85,B 0,C 180,E1 -28828.268,E2 -28828.268} C_VEL
LIN {X 0,Y 92.03,Z 517.555,A -85,B 0,C 180,E1 -28830.784,E2 -28830.784} C_VEL
LIN {X 0,Y 85.148,Z 524.088,A -85,B 0,C 180,E1 -28834.374,E2 -28834.374} C_VEL
LIN {X 0,Y 78.552,Z 529.689,A -85,B 0,C 180,E1 -28838.78,E2 -28838.78} C_VEL
LIN {X 0,Y 72.851,Z 534.086,A -85,B 0,C 180,E1 -28843.654,E2 -28843.654} C_VEL
LIN {X 0,Y 66.522,Z 538.413,A -85,B 0,C 180,E1 -28850.663,E2 -28850.663} C_VEL
LIN {X 0,Y 62.902,Z 540.782,A -85,B 0,C 180,E1 -28856.039,E2 -28856.039} C_VEL
LIN {X 0,Y 59.957,Z 542.587,A -85,B 0,C 180,E1 -28862.04,E2 -28862.04} C_VEL
LIN {X 0,Y 56.274,Z 545.053,A -85,B 0,C 180,E1 -28875.536,E2 -28875.536} C_VEL
LIN {X 0,Y 55.53,Z 545.652,A -85,B 0,C 180,E1 -28882.729,E2 -28882.729} C_VEL
LIN {X 0,Y 55.509,Z 545.816,A -85,B 0,C 180,E1 -28890,E2 -28890} C_VEL
LIN {X 0,Y 55.491,Z 545.651,A -85,B 0,C 180,E1 -28897.276,E2 -28897.276} C_VEL
LIN {X 0,Y 56.252,Z 545.052,A -85,B 0,C 180,E1 -28904.47,E2 -28904.47} C_VEL
LIN {X 0,Y 59.957,Z 542.587,A -85,B 0,C 180,E1 -28917.96,E2 -28917.96} C_VEL
LIN {X 0,Y 64.66,Z 539.631,A -85,B 0,C 180,E1 -28926.712,E2 -28926.712} C_VEL
LIN {X 0,Y 70.588,Z 535.638,A -85,B 0,C 180,E1 -28934.181,E2 -28934.181} C_VEL
LIN {X 0,Y 75.182,Z 532.426,A -85,B 0,C 180,E1 -28938.402,E2 -28938.402} C_VEL
LIN {X 0,Y 82.553,Z 526.401,A -85,B 0,C 180,E1 -28943.973,E2 -28943.973} C_VEL
LIN {X 0,Y 89.223,Z 520.305,A -85,B 0,C 180,E1 -28947.859,E2 -28947.859} C_VEL
LIN {X 0,Y 94.866,Z 514.609,A -85,B 0,C 180,E1 -28950.512,E2 -28950.512} C_VEL
LIN {X 0,Y 102.179,Z 506.062,A -85,B 0,C 180,E1 -28953.397,E2 -28953.397} C_VEL
LIN {X 0,Y 108.23,Z 497.891,A -85,B 0,C 180,E1 -28955.378,E2 -28955.378} C_VEL
LIN {X 0,Y 113.605,Z 489.387,A -85,B 0,C 180,E1 -28956.955,E2 -28956.955} C_VEL
LIN {X 0,Y 118.291,Z 480.679,A -85,B 0,C 180,E1 -28958.172,E2 -28958.172} C_VEL
LIN {X 0,Y 122.111,Z 472.223,A -85,B 0,C 180,E1 -28959.098,E2 -28959.098} C_VEL
LIN {X 0,Y 125.585,Z 462.831,A -85,B 0,C 180,E1 -28959.877,E2 -28959.877} C_VEL
LIN {X 0,Y 128.641,Z 452.048,A -85,B 0,C 180,E1 -28960.513,E2 -28960.513} C_VEL
LIN {X 0,Y 130.691,Z 441.497,A -85,B 0,C 180,E1 -28960.998,E2 -28960.998} C_VEL
LIN {X 0,Y 131.678,Z 433.874,A -85,B 0,C 180,E1 -28961.321,E2 -28961.321} C_VEL
LIN {X 0,Y 130.919,Z 431.015,A -85,B 0,C 180,E1 -28962.826,E2 -28962.826} C_VEL
LIN {X 0,Y 129.343,Z 426.978,A -85,B 0,C 180,E1 -28966.095,E2 -28966.095} C_VEL
LIN {X 0,Y 128.107,Z 424.048,A -85,B 0,C 180,E1 -28969.32,E2 -28969.32} C_VEL
LIN {X 0,Y 127.284,Z 421.925,A -85,B 0,C 180,E1 -28972.264,E2 -28972.264} C_VEL
LIN {X 0,Y 126.509,Z 418.334,A -85,B 0,C 180,E1 -28979.998,E2 -28979.998} C_VEL
LIN {X 0,Y 126.518,Z 419.658,A -85,B 0,C 180,E1 -28983.183,E2 -28983.183} C_VEL
LIN {X 0,Y 127.596,Z 422.607,A -85,B 0,C 180,E1 -28989.309,E2 -28989.309} C_VEL
LIN {X 0,Y 129.003,Z 426.17,A -85,B 0,C 180,E1 -28993.486,E2 -28993.486} C_VEL
LIN {X 0,Y 130.635,Z 430.216,A -85,B 0,C 180,E1 -28997.008,E2 -28997.008} C_VEL
LIN {X 0,Y 132.612,Z 435.911,A -85,B 0,C 180,E1 -29000.654,E2 -29000.654} C_VEL
LIN {X 0,Y 134.595,Z 443.301,A -85,B 0,C 180,E1 -29004.176,E2 -29004.176} C_VEL
LIN {X 0,Y 135.54,Z 449.815,A -85,B 0,C 180,E1 -29006.668,E2 -29006.668} C_VEL
LIN {X 0,Y 135.978,Z 456.723,A -85,B 0,C 180,E1 -29008.948,E2 -29008.948} C_VEL
LIN {X 0,Y 136.318,Z 464.894,A -85,B 0,C 180,E1 -29011.763,E2 -29011.763} C_VEL
LIN {X 0,Y 136.877,Z 474.884,A -85,B 0,C 180,E1 -29015.732,E2 -29015.732} C_VEL
LIN {X 0,Y 137.712,Z 483.451,A -85,B 0,C 180,E1 -29019.637,E2 -29019.637} C_VEL
LIN {X 0,Y 138.864,Z 490.61,A -85,B 0,C 180,E1 -29023.296,E2 -29023.296} C_VEL
LIN {X 0,Y 141.149,Z 499.209,A -85,B 0,C 180,E1 -29028.317,E2 -29028.317} C_VEL
LIN {X 0,Y 141.888,Z 501.138,A -85,B 0,C 180,E1 -29029.564,E2 -29029.564} C_VEL
LIN {X 0,Y 142.669,Z 504.555,A -85,B 0,C 180,E1 -29031.526,E2 -29031.526} C_VEL
LIN {X 0,Y 142.635,Z 510.387,A -85,B 0,C 180,E1 -29034.749,E2 -29034.749} C_VEL
LIN {X 0,Y 143.024,Z 515.666,A -85,B 0,C 180,E1 -29038.067,E2 -29038.067} C_VEL
LIN {X 0,Y 144.453,Z 518.184,A -85,B 0,C 180,E1 -29040.094,E2 -29040.094} C_VEL
LIN {X 0,Y 150.733,Z 523.523,A -85,B 0,C 180,E1 -29045.189,E2 -29045.189} C_VEL
LIN {X 0,Y 159.995,Z 528.643,A -85,B 0,C 180,E1 -29050.803,E2 -29050.803} C_VEL
LIN {X 0,Y 170.894,Z 532.508,A -85,B 0,C 180,E1 -29055.715,E2 -29055.715} C_VEL
LIN {X 0,Y 179.158,Z 534.583,A -85,B 0,C 180,E1 -29058.717,E2 -29058.717} C_VEL
LIN {X 0,Y 191.404,Z 536.667,A -85,B 0,C 180,E1 -29062.465,E2 -29062.465} C_VEL
LIN {X 0,Y 204.843,Z 538.006,A -85,B 0,C 180,E1 -29066.065,E2 -29066.065} C_VEL
LIN {X 0,Y 212.413,Z 538.371,A -85,B 0,C 180,E1 -29068.104,E2 -29068.104} C_VEL
LIN {X 0,Y 218.12,Z 538.393,A -85,B 0,C 180,E1 -29070,E2 -29070} C_VEL
LIN {X 0,Y 211.005,Z 538.307,A -85,B 0,C 180,E1 -29072.294,E2 -29072.294} C_VEL
LIN {X 0,Y 204.324,Z 537.966,A -85,B 0,C 180,E1 -29074.074,E2 -29074.074} C_VEL
LIN {X 0,Y 187.668,Z 536.107,A -85,B 0,C 180,E1 -29078.615,E2 -29078.615} C_VEL
LIN {X 0,Y 173.343,Z 533.175,A -85,B 0,C 180,E1 -29083.337,E2 -29083.337} C_VEL
LIN {X 0,Y 162.523,Z 529.656,A -85,B 0,C 180,E1 -29087.951,E2 -29087.951} C_VEL
LIN {X 0,Y 154.77,Z 526.034,A -85,B 0,C 180,E1 -29092.126,E2 -29092.126} C_VEL
LIN {X 0,Y 148.825,Z 522.117,A -85,B 0,C 180,E1 -29096.206,E2 -29096.206} C_VEL
LIN {X 0,Y 141.722,Z 515.212,A -85,B 0,C 180,E1 -29102.542,E2 -29102.542} C_VEL
LIN {X 0,Y 137.6,Z 508.744,A -85,B 0,C 180,E1 -29107.799,E2 -29107.799} C_VEL
LIN {X 0,Y 134.691,Z 501.446,A -85,B 0,C 180,E1 -29113.074,E2 -29113.074} C_VEL
LIN {X 0,Y 133.189,Z 494.209,A -85,B 0,C 180,E1 -29117.622,E2 -29117.622} C_VEL
LIN {X 0,Y 132.395,Z 486.953,A -85,B 0,C 180,E1 -29121.681,E2 -29121.681} C_VEL
LIN {X 0,Y 132.004,Z 478.358,A -85,B 0,C 180,E1 -29125.913,E2 -29125.913} C_VEL
LIN {X 0,Y 131.994,Z 468.457,A -85,B 0,C 180,E1 -29130.092,E2 -29130.092} C_VEL
LIN {X 0,Y 132.134,Z 458.544,A -85,B 0,C 180,E1 -29133.678,E2 -29133.678} C_VEL
LIN {X 0,Y 131.838,Z 450.394,A -85,B 0,C 180,E1 -29136.644,E2 -29136.644} C_VEL
LIN {X 0,Y 130.718,Z 443.163,A -85,B 0,C 180,E1 -29140.06,E2 -29140.06} C_VEL
LIN {X 0,Y 129.279,Z 437.662,A -85,B 0,C 180,E1 -29143.419,E2 -29143.419} C_VEL
LIN {X 0,Y 127.814,Z 433.221,A -85,B 0,C 180,E1 -29147.094,E2 -29147.094} C_VEL
LIN {X 0,Y 126.585,Z 429.815,A -85,B 0,C 180,E1 -29151.018,E2 -29151.018} C_VEL
LIN {X 0,Y 126.266,Z 428.879,A -85,B 0,C 180,E1 -29152.405,E2 -29152.405} C_VEL
LIN {X 0,Y 125.636,Z 425.449,A -85,B 0,C 180,E1 -29160.002,E2 -29160.002} C_VEL
LIN {X 0,Y 126.443,Z 429.347,A -85,B 0,C 180,E1 -29167.989,E2 -29167.989} C_VEL
LIN {X 0,Y 127.702,Z 432.898,A -85,B 0,C 180,E1 -29172.214,E2 -29172.214} C_VEL
LIN {X 0,Y 129.152,Z 437.118,A -85,B 0,C 180,E1 -29175.79,E2 -29175.79} C_VEL
LIN {X 0,Y 127.195,Z 448.647,A -85,B 0,C 180,E1 -29176.308,E2 -29176.308} C_VEL
LIN {X 0,Y 124.783,Z 458.084,A -85,B 0,C 180,E1 -29176.775,E2 -29176.775} C_VEL
LIN {X 0,Y 121.081,Z 468.825,A -85,B 0,C 180,E1 -29177.503,E2 -29177.503} C_VEL
LIN {X 0,Y 116.65,Z 478.854,A -85,B 0,C 180,E1 -29178.397,E2 -29178.397} C_VEL
LIN {X 0,Y 111.809,Z 487.842,A -85,B 0,C 180,E1 -29179.467,E2 -29179.467} C_VEL
LIN {X 0,Y 106.244,Z 496.563,A -85,B 0,C 180,E1 -29180.878,E2 -29180.878} C_VEL
LIN {X 0,Y 100.745,Z 503.95,A -85,B 0,C 180,E1 -29182.437,E2 -29182.437} C_VEL
LIN {X 0,Y 94.588,Z 511.163,A -85,B 0,C 180,E1 -29184.471,E2 -29184.471} C_VEL
LIN {X 0,Y 88.592,Z 517.361,A -85,B 0,C 180,E1 -29186.818,E2 -29186.818} C_VEL
LIN {X 0,Y 81.336,Z 523.894,A -85,B 0,C 180,E1 -29190.226,E2 -29190.226} C_VEL
LIN {X 0,Y 75.816,Z 528.396,A -85,B 0,C 180,E1 -29193.461,E2 -29193.461} C_VEL
LIN {X 0,Y 68.132,Z 533.891,A -85,B 0,C 180,E1 -29199.32,E2 -29199.32} C_VEL
LIN {X 0,Y 61.183,Z 538.218,A -85,B 0,C 180,E1 -29206.434,E2 -29206.434} C_VEL
LIN {X 0,Y 57.141,Z 540.588,A -85,B 0,C 180,E1 -29212.052,E2 -29212.052} C_VEL
LIN {X 0,Y 53.752,Z 542.392,A -85,B 0,C 180,E1 -29218.467,E2 -29218.467} C_VEL
LIN {X 0,Y 49.398,Z 544.858,A -85,B 0,C 180,E1 -29233.469,E2 -29233.469} C_VEL
LIN {X 0,Y 48.487,Z 545.458,A -85,B 0,C 180,E1 -29241.666,E2 -29241.666} C_VEL
LIN {X 0,Y 48.397,Z 545.622,A -85,B 0,C 180,E1 -29250,E2 -29250} C_VEL
LIN {X 0,Y 48.437,Z 545.457,A -85,B 0,C 180,E1 -29258.343,E2 -29258.343} C_VEL
LIN {X 0,Y 49.378,Z 544.858,A -85,B 0,C 180,E1 -29266.538,E2 -29266.538} C_VEL
LIN {X 0,Y 53.752,Z 542.392,A -85,B 0,C 180,E1 -29281.533,E2 -29281.533} C_VEL
LIN {X 0,Y 59.09,Z 539.436,A -85,B 0,C 180,E1 -29290.854,E2 -29290.854} C_VEL
LIN {X 0,Y 65.673,Z 535.444,A -85,B 0,C 180,E1 -29298.511,E2 -29298.511} C_VEL
LIN {X 0,Y 72.552,Z 530.787,A -85,B 0,C 180,E1 -29304.234,E2 -29304.234} C_VEL
LIN {X 0,Y 79.943,Z 525.05,A -85,B 0,C 180,E1 -29308.995,E2 -29308.995} C_VEL
LIN {X 0,Y 87.118,Z 518.736,A -85,B 0,C 180,E1 -29312.545,E2 -29312.545} C_VEL
LIN {X 0,Y 93.081,Z 512.789,A -85,B 0,C 180,E1 -29314.962,E2 -29314.962} C_VEL
LIN {X 0,Y 99.196,Z 505.868,A -85,B 0,C 180,E1 -29317.076,E2 -29317.076} C_VEL
LIN {X 0,Y 105.467,Z 497.697,A -85,B 0,C 180,E1 -29318.89,E2 -29318.89} C_VEL
LIN {X 0,Y 111.019,Z 489.194,A -85,B 0,C 180,E1 -29320.327,E2 -29320.327} C_VEL
LIN {X 0,Y 115.841,Z 480.485,A -85,B 0,C 180,E1 -29321.43,E2 -29321.43} C_VEL
LIN {X 0,Y 119.656,Z 472.296,A -85,B 0,C 180,E1 -29322.249,E2 -29322.249} C_VEL
LIN {X 0,Y 123.384,Z 462.463,A -85,B 0,C 180,E1 -29322.978,E2 -29322.978} C_VEL
LIN {X 0,Y 126.452,Z 451.837,A -85,B 0,C 180,E1 -29323.551,E2 -29323.551} C_VEL
LIN {X 0,Y 128.592,Z 441.079,A -85,B 0,C 180,E1 -29323.993,E2 -29323.993} C_VEL
LIN {X 0,Y 129.132,Z 437.121,A -85,B 0,C 180,E1 -29324.208,E2 -29324.208} C_VEL
LIN {X 0,Y 127.808,Z 433.211,A -85,B 0,C 180,E1 -29327.494,E2 -29327.494} C_VEL
LIN {X 0,Y 126.785,Z 430.442,A -85,B 0,C 180,E1 -29330.627,E2 -29330.627} C_VEL
LIN {X 0,Y 126.266,Z 428.849,A -85,B 0,C 180,E1 -29332.804,E2 -29332.804} C_VEL
LIN {X 0,Y 125.635,Z 425.457,A -85,B 0,C 180,E1 -29340.362,E2 -29340.362} C_VEL
LIN {X 0,Y 126.447,Z 429.35,A -85,B 0,C 180,E1 -29348.388,E2 -29348.388} C_VEL
LIN {X 0,Y 127.669,Z 432.846,A -85,B 0,C 180,E1 -29352.517,E2 -29352.517} C_VEL
LIN {X 0,Y 128.873,Z 436.452,A -85,B 0,C 180,E1 -29355.72,E2 -29355.72} C_VEL
LIN {X 0,Y 130.464,Z 442.103,A -85,B 0,C 180,E1 -29359.366,E2 -29359.366} C_VEL
LIN {X 0,Y 131.602,Z 448.858,A -85,B 0,C 180,E1 -29362.673,E2 -29362.673} C_VEL
LIN {X 0,Y 132.134,Z 455.26,A -85,B 0,C 180,E1 -29365.181,E2 -29365.181} C_VEL
LIN {X 0,Y 132.024,Z 466.159,A -85,B 0,C 180,E1 -29369.027,E2 -29369.027} C_VEL
LIN {X 0,Y 131.957,Z 475.504,A -85,B 0,C 180,E1 -29372.815,E2 -29372.815} C_VEL
LIN {X 0,Y 132.2,Z 483.842,A -85,B 0,C 180,E1 -29376.73,E2 -29376.73} C_VEL
LIN {X 0,Y 132.876,Z 492.113,A -85,B 0,C 180,E1 -29381.142,E2 -29381.142} C_VEL
LIN {X 0,Y 134.312,Z 499.792,A -85,B 0,C 180,E1 -29385.849,E2 -29385.849} C_VEL
LIN {X 0,Y 136.575,Z 506.529,A -85,B 0,C 180,E1 -29390.521,E2 -29390.521} C_VEL
LIN {X 0,Y 140.267,Z 513.183,A -85,B 0,C 180,E1 -29395.741,E2 -29395.741} C_VEL
LIN {X 0,Y 144.453,Z 518.184,A -85,B 0,C 180,E1 -29400.094,E2 -29400.094} C_VEL
LIN {X 0,Y 146.072,Z 520.595,A -85,B 0,C 180,E1 -29402.14,E2 -29402.14} C_VEL
LIN {X 0,Y 149.089,Z 527.919,A -85,B 0,C 180,E1 -29408.364,E2 -29408.364} C_VEL
LIN {X 0,Y 151.21,Z 529.643,A -85,B 0,C 180,E1 -29410.334,E2 -29410.334} C_VEL
LIN {X 0,Y 152.188,Z 530.122,A -85,B 0,C 180,E1 -29410.945,E2 -29410.945} C_VEL
LIN {X 0,Y 165.739,Z 534.495,A -85,B 0,C 180,E1 -29417.23,E2 -29417.23} C_VEL
LIN {X 0,Y 177.694,Z 536.73,A -85,B 0,C 180,E1 -29421.398,E2 -29421.398} C_VEL
LIN {X 0,Y 193.436,Z 538.319,A -85,B 0,C 180,E1 -29425.833,E2 -29425.833} C_VEL
LIN {X 0,Y 203.874,Z 538.709,A -85,B 0,C 180,E1 -29428.541,E2 -29428.541} C_VEL
LIN {X 0,Y 208.92,Z 538.639,A -85,B 0,C 180,E1 -29430,E2 -29430} C_VEL
LIN {X 0,Y 201.809,Z 538.659,A -85,B 0,C 180,E1 -29431.996,E2 -29431.996} C_VEL
LIN {X 0,Y 190.459,Z 538.121,A -85,B 0,C 180,E1 -29434.941,E2 -29434.941} C_VEL
LIN {X 0,Y 175.796,Z 536.428,A -85,B 0,C 180,E1 -29439.202,E2 -29439.202} C_VEL
LIN {X 0,Y 165.74,Z 534.494,A -85,B 0,C 180,E1 -29442.771,E2 -29442.771} C_VEL
LIN {X 0,Y 152.647,Z 530.32,A -85,B 0,C 180,E1 -29448.801,E2 -29448.801} C_VEL
LIN {X 0,Y 145.401,Z 526.702,A -85,B 0,C 180,E1 -29453.315,E2 -29453.315} C_VEL
LIN {X 0,Y 139.359,Z 522.348,A -85,B 0,C 180,E1 -29458.177,E2 -29458.177} C_VEL
LIN {X 0,Y 134.539,Z 517.246,A -85,B 0,C 180,E1 -29463.304,E2 -29463.304} C_VEL
LIN {X 0,Y 130.316,Z 509.849,A -85,B 0,C 180,E1 -29469.785,E2 -29469.785} C_VEL
LIN {X 0,Y 128.076,Z 502.362,A -85,B 0,C 180,E1 -29475.507,E2 -29475.507} C_VEL
LIN {X 0,Y 127.131,Z 494.462,A -85,B 0,C 180,E1 -29480.708,E2 -29480.708} C_VEL
LIN {X 0,Y 127.031,Z 486.058,A -85,B 0,C 180,E1 -29485.457,E2 -29485.457} C_VEL
LIN {X 0,Y 127.34,Z 478.145,A -85,B 0,C 180,E1 -29489.37,E2 -29489.37} C_VEL
LIN {X 0,Y 127.969,Z 468.69,A -85,B 0,C 180,E1 -29493.392,E2 -29493.392} C_VEL
LIN {X 0,Y 128.607,Z 459.148,A -85,B 0,C 180,E1 -29496.908,E2 -29496.908} C_VEL
LIN {X 0,Y 128.616,Z 454.013,A -85,B 0,C 180,E1 -29499.03,E2 -29499.03} C_VEL
LIN {X 0,Y 127.918,Z 447.715,A -85,B 0,C 180,E1 -29502.207,E2 -29502.207} C_VEL
LIN {X 0,Y 127.046,Z 442.659,A -85,B 0,C 180,E1 -29505.587,E2 -29505.587} C_VEL
LIN {X 0,Y 125.978,Z 438.563,A -85,B 0,C 180,E1 -29509.353,E2 -29509.353} C_VEL
LIN {X 0,Y 125.18,Z 435.696,A -85,B 0,C 180,E1 -29513.15,E2 -29513.15} C_VEL
LIN {X 0,Y 124.744,Z 432.711,A -85,B 0,C 180,E1 -29520.002,E2 -29520.002} C_VEL
LIN {X 0,Y 125.336,Z 436.216,A -85,B 0,C 180,E1 -29527.25,E2 -29527.25} C_VEL
LIN {X 0,Y 126.338,Z 439.713,A -85,B 0,C 180,E1 -29531.432,E2 -29531.432} C_VEL
LIN {X 0,Y 126.758,Z 441.302,A -85,B 0,C 180,E1 -29532.881,E2 -29532.881} C_VEL
LIN {X 0,Y 124.498,Z 452.215,A -85,B 0,C 180,E1 -29533.352,E2 -29533.352} C_VEL
LIN {X 0,Y 120.592,Z 465.058,A -85,B 0,C 180,E1 -29534.005,E2 -29534.005} C_VEL
LIN {X 0,Y 115.432,Z 477.029,A -85,B 0,C 180,E1 -29534.869,E2 -29534.869} C_VEL
LIN {X 0,Y 110.474,Z 486.298,A -85,B 0,C 180,E1 -29535.809,E2 -29535.809} C_VEL
LIN {X 0,Y 104.737,Z 495.235,A -85,B 0,C 180,E1 -29537.025,E2 -29537.025} C_VEL
LIN {X 0,Y 98.252,Z 503.756,A -85,B 0,C 180,E1 -29538.603,E2 -29538.603} C_VEL
LIN {X 0,Y 91.874,Z 510.969,A -85,B 0,C 180,E1 -29540.437,E2 -29540.437} C_VEL
LIN {X 0,Y 85.606,Z 517.165,A -85,B 0,C 180,E1 -29542.547,E2 -29542.547} C_VEL
LIN {X 0,Y 77.991,Z 523.699,A -85,B 0,C 180,E1 -29545.696,E2 -29545.696} C_VEL
LIN {X 0,Y 72.114,Z 528.2,A -85,B 0,C 180,E1 -29548.707,E2 -29548.707} C_VEL
LIN {X 0,Y 63.858,Z 533.697,A -85,B 0,C 180,E1 -29554.37,E2 -29554.37} C_VEL
LIN {X 0,Y 56.226,Z 538.023,A -85,B 0,C 180,E1 -29561.414,E2 -29561.414} C_VEL
LIN {X 0,Y 51.717,Z 540.393,A -85,B 0,C 180,E1 -29567.199,E2 -29567.199} C_VEL
LIN {X 0,Y 47.812,Z 542.197,A -85,B 0,C 180,E1 -29573.988,E2 -29573.988} C_VEL
LIN {X 0,Y 42.615,Z 544.664,A -85,B 0,C 180,E1 -29590.742,E2 -29590.742} C_VEL
LIN {X 0,Y 41.458,Z 545.264,A -85,B 0,C 180,E1 -29600.24,E2 -29600.24} C_VEL
LIN {X 0,Y 41.302,Z 545.428,A -85,B 0,C 180,E1 -29610,E2 -29610} C_VEL
LIN {X 0,Y 41.419,Z 545.263,A -85,B 0,C 180,E1 -29619.769,E2 -29619.769} C_VEL
LIN {X 0,Y 42.599,Z 544.663,A -85,B 0,C 180,E1 -29629.266,E2 -29629.266} C_VEL
LIN {X 0,Y 47.812,Z 542.197,A -85,B 0,C 180,E1 -29646.012,E2 -29646.012} C_VEL
LIN {X 0,Y 53.899,Z 539.241,A -85,B 0,C 180,E1 -29655.819,E2 -29655.819} C_VEL
LIN {X 0,Y 61.194,Z 535.25,A -85,B 0,C 180,E1 -29663.505,E2 -29663.505} C_VEL
LIN {X 0,Y 69.512,Z 529.99,A -85,B 0,C 180,E1 -29669.63,E2 -29669.63} C_VEL
LIN {X 0,Y 76.514,Z 524.855,A -85,B 0,C 180,E1 -29673.578,E2 -29673.578} C_VEL
LIN {X 0,Y 84.077,Z 518.542,A -85,B 0,C 180,E1 -29676.848,E2 -29676.848} C_VEL
LIN {X 0,Y 90.302,Z 512.595,A -85,B 0,C 180,E1 -29679.053,E2 -29679.053} C_VEL
LIN {X 0,Y 96.645,Z 505.673,A -85,B 0,C 180,E1 -29680.968,E2 -29680.968} C_VEL
LIN {X 0,Y 103.121,Z 497.503,A -85,B 0,C 180,E1 -29682.576,E2 -29682.576} C_VEL
LIN {X 0,Y 108.834,Z 489,A -85,B 0,C 180,E1 -29683.849,E2 -29683.849} C_VEL
LIN {X 0,Y 113.779,Z 480.291,A -85,B 0,C 180,E1 -29684.822,E2 -29684.822} C_VEL
LIN {X 0,Y 118.232,Z 470.818,A -85,B 0,C 180,E1 -29685.606,E2 -29685.606} C_VEL
LIN {X 0,Y 121.866,Z 461.131,A -85,B 0,C 180,E1 -29686.237,E2 -29686.237} C_VEL
LIN {X 0,Y 124.802,Z 450.937,A -85,B 0,C 180,E1 -29686.699,E2 -29686.699} C_VEL
LIN {X 0,Y 126.73,Z 441.286,A -85,B 0,C 180,E1 -29687.116,E2 -29687.116} C_VEL
LIN {X 0,Y 125.68,Z 437.565,A -85,B 0,C 180,E1 -29690.95,E2 -29690.95} C_VEL
LIN {X 0,Y 125.118,Z 435.53,A -85,B 0,C 180,E1 -29693.953,E2 -29693.953} C_VEL
LIN {X 0,Y 124.747,Z 432.691,A -85,B 0,C 180,E1 -29700.402,E2 -29700.402} C_VEL
LIN {X 0,Y 125.321,Z 436.376,A -85,B 0,C 180,E1 -29707.855,E2 -29707.855} C_VEL
LIN {X 0,Y 126.185,Z 439.532,A -85,B 0,C 180,E1 -29711.646,E2 -29711.646} C_VEL
LIN {X 0,Y 127.306,Z 443.881,A -85,B 0,C 180,E1 -29715.303,E2 -29715.303} C_VEL
LIN {X 0,Y 128.058,Z 448.804,A -85,B 0,C 180,E1 -29718.393,E2 -29718.393} C_VEL
LIN {X 0,Y 128.606,Z 454.046,A -85,B 0,C 180,E1 -29720.972,E2 -29720.972} C_VEL
LIN {X 0,Y 128.561,Z 460.843,A -85,B 0,C 180,E1 -29723.707,E2 -29723.707} C_VEL
LIN {X 0,Y 127.723,Z 472.936,A -85,B 0,C 180,E1 -29728.311,E2 -29728.311} C_VEL
LIN {X 0,Y 127.125,Z 483.068,A -85,B 0,C 180,E1 -29732.985,E2 -29732.985} C_VEL
LIN {X 0,Y 127.075,Z 491.372,A -85,B 0,C 180,E1 -29737.469,E2 -29737.469} C_VEL
LIN {X 0,Y 127.77,Z 500.047,A -85,B 0,C 180,E1 -29742.927,E2 -29742.927} C_VEL
LIN {X 0,Y 129.419,Z 507.326,A -85,B 0,C 180,E1 -29748.217,E2 -29748.217} C_VEL
LIN {X 0,Y 131.946,Z 513.162,A -85,B 0,C 180,E1 -29753.028,E2 -29753.028} C_VEL
LIN {X 0,Y 136.628,Z 519.576,A -85,B 0,C 180,E1 -29759.044,E2 -29759.044} C_VEL
LIN {X 0,Y 141.326,Z 523.929,A -85,B 0,C 180,E1 -29763.521,E2 -29763.521} C_VEL
LIN {X 0,Y 149.929,Z 529.115,A -85,B 0,C 180,E1 -29769.633,E2 -29769.633} C_VEL
LIN {X 0,Y 152.188,Z 530.122,A -85,B 0,C 180,E1 -29770.945,E2 -29770.945} C_VEL
LIN {X 0,Y 154.927,Z 531.704,A -85,B 0,C 180,E1 -29772.822,E2 -29772.822} C_VEL
LIN {X 0,Y 159.827,Z 535.16,A -85,B 0,C 180,E1 -29777.383,E2 -29777.383} C_VEL
LIN {X 0,Y 163.536,Z 536.547,A -85,B 0,C 180,E1 -29779.791,E2 -29779.791} C_VEL
LIN {X 0,Y 166.036,Z 537.023,A -85,B 0,C 180,E1 -29780.827,E2 -29780.827} C_VEL
LIN {X 0,Y 183.172,Z 538.705,A -85,B 0,C 180,E1 -29785.989,E2 -29785.989} C_VEL
LIN {X 0,Y 190.57,Z 538.965,A -85,B 0,C 180,E1 -29787.887,E2 -29787.887} C_VEL
LIN {X 0,Y 198.961,Z 538.906,A -85,B 0,C 180,E1 -29790,E2 -29790} C_VEL
LIN {X 0,Y 189.902,Z 538.945,A -85,B 0,C 180,E1 -29792.282,E2 -29792.282} C_VEL
LIN {X 0,Y 176.609,Z 538.264,A -85,B 0,C 180,E1 -29795.831,E2 -29795.831} C_VEL
LIN {X 0,Y 164.066,Z 536.747,A -85,B 0,C 180,E1 -29799.866,E2 -29799.866} C_VEL
LIN {X 0,Y 152.519,Z 534.256,A -85,B 0,C 180,E1 -29804.616,E2 -29804.616} C_VEL
LIN {X 0,Y 142.241,Z 530.616,A -85,B 0,C 180,E1 -29810.234,E2 -29810.234} C_VEL
LIN {X 0,Y 135.93,Z 527.143,A -85,B 0,C 180,E1 -29814.905,E2 -29814.905} C_VEL
LIN {X 0,Y 130.301,Z 522.61,A -85,B 0,C 180,E1 -29820.35,E2 -29820.35} C_VEL
LIN {X 0,Y 126.112,Z 517.202,A -85,B 0,C 180,E1 -29826.096,E2 -29826.096} C_VEL
LIN {X 0,Y 123.25,Z 510.7,A -85,B 0,C 180,E1 -29832.161,E2 -29832.161} C_VEL
LIN {X 0,Y 121.944,Z 504.184,A -85,B 0,C 180,E1 -29837.476,E2 -29837.476} C_VEL
LIN {X 0,Y 121.595,Z 495.807,A -85,B 0,C 180,E1 -29843.316,E2 -29843.316} C_VEL
LIN {X 0,Y 122.118,Z 487.69,A -85,B 0,C 180,E1 -29848.128,E2 -29848.128} C_VEL
LIN {X 0,Y 123.073,Z 479.357,A -85,B 0,C 180,E1 -29852.366,E2 -29852.366} C_VEL
LIN {X 0,Y 124.404,Z 469.256,A -85,B 0,C 180,E1 -29856.708,E2 -29856.708} C_VEL
LIN {X 0,Y 125.297,Z 462.032,A -85,B 0,C 180,E1 -29859.523,E2 -29859.523} C_VEL
LIN {X 0,Y 125.435,Z 456.057,A -85,B 0,C 180,E1 -29862.264,E2 -29862.264} C_VEL
LIN {X 0,Y 125.157,Z 451.159,A -85,B 0,C 180,E1 -29865.157,E2 -29865.157} C_VEL
LIN {X 0,Y 124.555,Z 446.564,A -85,B 0,C 180,E1 -29868.818,E2 -29868.818} C_VEL
LIN {X 0,Y 124.036,Z 443.505,A -85,B 0,C 180,E1 -29872.473,E2 -29872.473} C_VEL
LIN {X 0,Y 123.761,Z 442.176,A -85,B 0,C 180,E1 -29874.707,E2 -29874.707} C_VEL
LIN {X 0,Y 123.681,Z 439.914,A -85,B 0,C 180,E1 -29880.002,E2 -29880.002} C_VEL
LIN {X 0,Y 124.001,Z 443.029,A -85,B 0,C 180,E1 -29886.51,E2 -29886.51} C_VEL
LIN {X 0,Y 124.552,Z 445.724,A -85,B 0,C 180,E1 -29889.86,E2 -29889.86} C_VEL
LIN {X 0,Y 121.448,Z 457.696,A -85,B 0,C 180,E1 -29890.348,E2 -29890.348} C_VEL
LIN {X 0,Y 117.67,Z 468.254,A -85,B 0,C 180,E1 -29890.881,E2 -29890.881} C_VEL
LIN {X 0,Y 113.815,Z 476.835,A -85,B 0,C 180,E1 -29891.407,E2 -29891.407} C_VEL
LIN {X 0,Y 108.758,Z 486.105,A -85,B 0,C 180,E1 -29892.214,E2 -29892.214} C_VEL
LIN {X 0,Y 102.884,Z 495.041,A -85,B 0,C 180,E1 -29893.247,E2 -29893.247} C_VEL
LIN {X 0,Y 96.222,Z 503.562,A -85,B 0,C 180,E1 -29894.592,E2 -29894.592} C_VEL
LIN {X 0,Y 89.643,Z 510.775,A -85,B 0,C 180,E1 -29896.182,E2 -29896.182} C_VEL
LIN {X 0,Y 83.134,Z 516.971,A -85,B 0,C 180,E1 -29898.005,E2 -29898.005} C_VEL
LIN {X 0,Y 75.181,Z 523.505,A -85,B 0,C 180,E1 -29900.806,E2 -29900.806} C_VEL
LIN {X 0,Y 66.931,Z 529.297,A -85,B 0,C 180,E1 -29904.548,E2 -29904.548} C_VEL
LIN {X 0,Y 60.113,Z 533.502,A -85,B 0,C 180,E1 -29908.738,E2 -29908.738} C_VEL
LIN {X 0,Y 51.773,Z 537.828,A -85,B 0,C 180,E1 -29915.466,E2 -29915.466} C_VEL
LIN {X 0,Y 46.73,Z 540.198,A -85,B 0,C 180,E1 -29921.24,E2 -29921.24} C_VEL
LIN {X 0,Y 42.248,Z 542.002,A -85,B 0,C 180,E1 -29928.288,E2 -29928.288} C_VEL
LIN {X 0,Y 35.973,Z 544.469,A -85,B 0,C 180,E1 -29947.001,E2 -29947.001} C_VEL
LIN {X 0,Y 34.479,Z 545.07,A -85,B 0,C 180,E1 -29958.239,E2 -29958.239} C_VEL
LIN {X 0,Y 34.189,Z 545.234,A -85,B 0,C 180,E1 -29970,E2 -29970} C_VEL
LIN {X 0,Y 34.447,Z 545.069,A -85,B 0,C 180,E1 -29981.772,E2 -29981.772} C_VEL
LIN {X 0,Y 35.961,Z 544.469,A -85,B 0,C 180,E1 -29993.008,E2 -29993.008} C_VEL
LIN {X 0,Y 42.248,Z 542.002,A -85,B 0,C 180,E1 -30011.713,E2 -30011.713} C_VEL
LIN {X 0,Y 49.198,Z 539.047,A -85,B 0,C 180,E1 -30021.782,E2 -30021.782} C_VEL
LIN {X 0,Y 57.252,Z 535.056,A -85,B 0,C 180,E1 -30029.234,E2 -30029.234} C_VEL
LIN {X 0,Y 66.288,Z 529.728,A -85,B 0,C 180,E1 -30035.036,E2 -30035.036} C_VEL
LIN {X 0,Y 73.617,Z 524.66,A -85,B 0,C 180,E1 -30038.556,E2 -30038.556} C_VEL
LIN {X 0,Y 81.543,Z 518.347,A -85,B 0,C 180,E1 -30041.45,E2 -30041.45} C_VEL
LIN {X 0,Y 88.013,Z 512.401,A -85,B 0,C 180,E1 -30043.376,E2 -30043.376} C_VEL
LIN {X 0,Y 94.563,Z 505.479,A -85,B 0,C 180,E1 -30045.049,E2 -30045.049} C_VEL
LIN {X 0,Y 101.22,Z 497.309,A -85,B 0,C 180,E1 -30046.417,E2 -30046.417} C_VEL
LIN {X 0,Y 107.076,Z 488.806,A -85,B 0,C 180,E1 -30047.503,E2 -30047.503} C_VEL
LIN {X 0,Y 112.129,Z 480.097,A -85,B 0,C 180,E1 -30048.326,E2 -30048.326} C_VEL
LIN {X 0,Y 116.468,Z 471.105,A -85,B 0,C 180,E1 -30048.955,E2 -30048.955} C_VEL
LIN {X 0,Y 120.378,Z 460.937,A -85,B 0,C 180,E1 -30049.513,E2 -30049.513} C_VEL
LIN {X 0,Y 123.473,Z 450.292,A -85,B 0,C 180,E1 -30049.92,E2 -30049.92} C_VEL
LIN {X 0,Y 124.546,Z 445.751,A -85,B 0,C 180,E1 -30050.139,E2 -30050.139} C_VEL
LIN {X 0,Y 123.944,Z 442.681,A -85,B 0,C 180,E1 -30053.895,E2 -30053.895} C_VEL
LIN {X 0,Y 123.639,Z 439.905,A -85,B 0,C 180,E1 -30060.405,E2 -30060.405} C_VEL
LIN {X 0,Y 123.989,Z 443.164,A -85,B 0,C 180,E1 -30067.121,E2 -30067.121} C_VEL
LIN {X 0,Y 124.551,Z 446.582,A -85,B 0,C 180,E1 -30071.183,E2 -30071.183} C_VEL
LIN {X 0,Y 125.211,Z 451.621,A -85,B 0,C 180,E1 -30075.148,E2 -30075.148} C_VEL
LIN {X 0,Y 125.423,Z 456.058,A -85,B 0,C 180,E1 -30077.719,E2 -30077.719} C_VEL
LIN {X 0,Y 125.299,Z 462.043,A -85,B 0,C 180,E1 -30080.484,E2 -30080.484} C_VEL
LIN {X 0,Y 123.807,Z 473.924,A -85,B 0,C 180,E1 -30085.194,E2 -30085.194} C_VEL
LIN {X 0,Y 122.59,Z 483.386,A -85,B 0,C 180,E1 -30089.611,E2 -30089.611} C_VEL
LIN {X 0,Y 121.784,Z 492.45,A -85,B 0,C 180,E1 -30094.644,E2 -30094.644} C_VEL
LIN {X 0,Y 121.628,Z 499.937,A -85,B 0,C 180,E1 -30099.463,E2 -30099.463} C_VEL
LIN {X 0,Y 122.458,Z 507.627,A -85,B 0,C 180,E1 -30105.265,E2 -30105.265} C_VEL
LIN {X 0,Y 124.343,Z 513.767,A -85,B 0,C 180,E1 -30110.61,E2 -30110.61} C_VEL
LIN {X 0,Y 127.935,Z 519.856,A -85,B 0,C 180,E1 -30116.679,E2 -30116.679} C_VEL
LIN {X 0,Y 133.803,Z 525.619,A -85,B 0,C 180,E1 -30123.239,E2 -30123.239} C_VEL
LIN {X 0,Y 140.007,Z 529.5,A -85,B 0,C 180,E1 -30128.221,E2 -30128.221} C_VEL
LIN {X 0,Y 148.731,Z 533.123,A -85,B 0,C 180,E1 -30133.53,E2 -30133.53} C_VEL
LIN {X 0,Y 158.149,Z 535.63,A -85,B 0,C 180,E1 -30137.86,E2 -30137.86} C_VEL
LIN {X 0,Y 166.036,Z 537.023,A -85,B 0,C 180,E1 -30140.827,E2 -30140.827} C_VEL
LIN {X 0,Y 169.77,Z 537.704,A -85,B 0,C 180,E1 -30142.376,E2 -30142.376} C_VEL
LIN {X 0,Y 174.884,Z 538.756,A -85,B 0,C 180,E1 -30145.18,E2 -30145.18} C_VEL
LIN {X 0,Y 179.124,Z 539.22,A -85,B 0,C 180,E1 -30147.353,E2 -30147.353} C_VEL
LIN {X 0,Y 182.995,Z 539.312,A -85,B 0,C 180,E1 -30148.772,E2 -30148.772} C_VEL
LIN {X 0,Y 184.478,Z 539.278,A -85,B 0,C 180,E1 -30149.179,E2 -30149.179} C_VEL
LIN {X 0,Y 187.826,Z 539.204,A -85,B 0,C 180,E1 -30150,E2 -30150} C_VEL
LIN {X 0,Y 175.936,Z 539.194,A -85,B 0,C 180,E1 -30152.997,E2 -30152.997} C_VEL
LIN {X 0,Y 160.819,Z 538.177,A -85,B 0,C 180,E1 -30157.533,E2 -30157.533} C_VEL
LIN {X 0,Y 150.577,Z 536.677,A -85,B 0,C 180,E1 -30161.443,E2 -30161.443} C_VEL
LIN {X 0,Y 144.893,Z 535.507,A -85,B 0,C 180,E1 -30164.054,E2 -30164.054} C_VEL
LIN {X 0,Y 134.645,Z 532.146,A -85,B 0,C 180,E1 -30170.031,E2 -30170.031} C_VEL
LIN {X 0,Y 126.289,Z 527.305,A -85,B 0,C 180,E1 -30177.08,E2 -30177.08} C_VEL
LIN {X 0,Y 121.437,Z 522.735,A -85,B 0,C 180,E1 -30182.972,E2 -30182.972} C_VEL
LIN {X 0,Y 118.041,Z 517.14,A -85,B 0,C 180,E1 -30189.288,E2 -30189.288} C_VEL
LIN {X 0,Y 116.198,Z 510.416,A -85,B 0,C 180,E1 -30195.828,E2 -30195.828} C_VEL
LIN {X 0,Y 115.879,Z 502.866,A -85,B 0,C 180,E1 -30202.039,E2 -30202.039} C_VEL
LIN {X 0,Y 116.61,Z 494.951,A -85,B 0,C 180,E1 -30207.538,E2 -30207.538} C_VEL
LIN {X 0,Y 117.633,Z 488.496,A -85,B 0,C 180,E1 -30211.45,E2 -30211.45} C_VEL
LIN {X 0,Y 119.399,Z 479.311,A -85,B 0,C 180,E1 -30216.132,E2 -30216.132} C_VEL
LIN {X 0,Y 121.252,Z 469.975,A -85,B 0,C 180,E1 -30220.148,E2 -30220.148} C_VEL
LIN {X 0,Y 122.298,Z 463.702,A -85,B 0,C 180,E1 -30222.816,E2 -30222.816} C_VEL
LIN {X 0,Y 122.554,Z 458.083,A -85,B 0,C 180,E1 -30225.896,E2 -30225.896} C_VEL
LIN {X 0,Y 122.567,Z 454.671,A -85,B 0,C 180,E1 -30228.423,E2 -30228.423} C_VEL
LIN {X 0,Y 122.313,Z 451.061,A -85,B 0,C 180,E1 -30231.951,E2 -30231.951} C_VEL
LIN {X 0,Y 122.12,Z 449.027,A -85,B 0,C 180,E1 -30235.05,E2 -30235.05} C_VEL
LIN {X 0,Y 122.237,Z 447.038,A -85,B 0,C 180,E1 -30240.002,E2 -30240.002} C_VEL
LIN {X 0,Y 122.26,Z 449.752,A -85,B 0,C 180,E1 -30245.775,E2 -30245.775} C_VEL
LIN {X 0,Y 122.326,Z 450.456,A -85,B 0,C 180,E1 -30246.754,E2 -30246.754} C_VEL
LIN {X 0,Y 119.779,Z 459.29,A -85,B 0,C 180,E1 -30247.09,E2 -30247.09} C_VEL
LIN {X 0,Y 116.223,Z 468.797,A -85,B 0,C 180,E1 -30247.483,E2 -30247.483} C_VEL
LIN {X 0,Y 111.771,Z 478.273,A -85,B 0,C 180,E1 -30247.981,E2 -30247.981} C_VEL
LIN {X 0,Y 106.622,Z 487.261,A -85,B 0,C 180,E1 -30248.62,E2 -30248.62} C_VEL
LIN {X 0,Y 100.64,Z 495.981,A -85,B 0,C 180,E1 -30249.47,E2 -30249.47} C_VEL
LIN {X 0,Y 94.684,Z 503.368,A -85,B 0,C 180,E1 -30250.432,E2 -30250.432} C_VEL
LIN {X 0,Y 87.927,Z 510.581,A -85,B 0,C 180,E1 -30251.73,E2 -30251.73} C_VEL
LIN {X 0,Y 81.218,Z 516.777,A -85,B 0,C 180,E1 -30253.229,E2 -30253.229} C_VEL
LIN {X 0,Y 72.954,Z 523.31,A -85,B 0,C 180,E1 -30255.565,E2 -30255.565} C_VEL
LIN {X 0,Y 66.444,Z 527.81,A -85,B 0,C 180,E1 -30257.837,E2 -30257.837} C_VEL
LIN {X 0,Y 57.022,Z 533.307,A -85,B 0,C 180,E1 -30262.43,E2 -30262.43} C_VEL
LIN {X 0,Y 47.98,Z 537.633,A -85,B 0,C 180,E1 -30268.497,E2 -30268.497} C_VEL
LIN {X 0,Y 42.369,Z 540.004,A -85,B 0,C 180,E1 -30273.968,E2 -30273.968} C_VEL
LIN {X 0,Y 37.224,Z 541.807,A -85,B 0,C 180,E1 -30280.957,E2 -30280.957} C_VEL
LIN {X 0,Y 29.535,Z 544.274,A -85,B 0,C 180,E1 -30301.582,E2 -30301.582} C_VEL
LIN {X 0,Y 27.547,Z 544.875,A -85,B 0,C 180,E1 -30315.219,E2 -30315.219} C_VEL
LIN {X 0,Y 27.077,Z 545.04,A -85,B 0,C 180,E1 -30330,E2 -30330} C_VEL
LIN {X 0,Y 27.521,Z 544.875,A -85,B 0,C 180,E1 -30344.795,E2 -30344.795} C_VEL
LIN {X 0,Y 29.525,Z 544.274,A -85,B 0,C 180,E1 -30358.428,E2 -30358.428} C_VEL
LIN {X 0,Y 37.224,Z 541.807,A -85,B 0,C 180,E1 -30379.043,E2 -30379.043} C_VEL
LIN {X 0,Y 45.137,Z 538.852,A -85,B 0,C 180,E1 -30388.909,E2 -30388.909} C_VEL
LIN {X 0,Y 53.961,Z 534.862,A -85,B 0,C 180,E1 -30395.737,E2 -30395.737} C_VEL
LIN {X 0,Y 61.866,Z 530.589,A -85,B 0,C 180,E1 -30400.07,E2 -30400.07} C_VEL
LIN {X 0,Y 69.696,Z 525.621,A -85,B 0,C 180,E1 -30403.323,E2 -30403.323} C_VEL
LIN {X 0,Y 77.905,Z 519.528,A -85,B 0,C 180,E1 -30405.874,E2 -30405.874} C_VEL
LIN {X 0,Y 84.566,Z 513.832,A -85,B 0,C 180,E1 -30407.549,E2 -30407.549} C_VEL
LIN {X 0,Y 92.982,Z 505.285,A -85,B 0,C 180,E1 -30409.289,E2 -30409.289} C_VEL
LIN {X 0,Y 99.79,Z 497.115,A -85,B 0,C 180,E1 -30410.391,E2 -30410.391} C_VEL
LIN {X 0,Y 105.765,Z 488.612,A -85,B 0,C 180,E1 -30411.268,E2 -30411.268} C_VEL
LIN {X 0,Y 110.911,Z 479.903,A -85,B 0,C 180,E1 -30411.92,E2 -30411.92} C_VEL
LIN {X 0,Y 115.585,Z 470.295,A -85,B 0,C 180,E1 -30412.439,E2 -30412.439} C_VEL
LIN {X 0,Y 119.23,Z 460.932,A -85,B 0,C 180,E1 -30412.851,E2 -30412.851} C_VEL
LIN {X 0,Y 122.322,Z 450.483,A -85,B 0,C 180,E1 -30413.233,E2 -30413.233} C_VEL
LIN {X 0,Y 122.157,Z 448.859,A -85,B 0,C 180,E1 -30415.874,E2 -30415.874} C_VEL
LIN {X 0,Y 122.241,Z 447.023,A -85,B 0,C 180,E1 -30419.998,E2 -30419.998} C_VEL
LIN {X 0,Y 122.184,Z 449.724,A -85,B 0,C 180,E1 -30426.19,E2 -30426.19} C_VEL
LIN {X 0,Y 122.473,Z 452.796,A -85,B 0,C 180,E1 -30429.911,E2 -30429.911} C_VEL
LIN {X 0,Y 122.585,Z 456.786,A -85,B 0,C 180,E1 -30433.256,E2 -30433.256} C_VEL
LIN {X 0,Y 122.378,Z 462.714,A -85,B 0,C 180,E1 -30436.685,E2 -30436.685} C_VEL
LIN {X 0,Y 121.75,Z 467.215,A -85,B 0,C 180,E1 -30438.767,E2 -30438.767} C_VEL
LIN {X 0,Y 120.067,Z 475.949,A -85,B 0,C 180,E1 -30442.359,E2 -30442.359} C_VEL
LIN {X 0,Y 118.53,Z 483.787,A -85,B 0,C 180,E1 -30446.07,E2 -30446.07} C_VEL
LIN {X 0,Y 117.087,Z 491.748,A -85,B 0,C 180,E1 -30450.441,E2 -30450.441} C_VEL
LIN {X 0,Y 116.004,Z 500.608,A -85,B 0,C 180,E1 -30456.291,E2 -30456.291} C_VEL
LIN {X 0,Y 115.97,Z 507.653,A -85,B 0,C 180,E1 -30461.804,E2 -30461.804} C_VEL
LIN {X 0,Y 117,Z 514.032,A -85,B 0,C 180,E1 -30467.591,E2 -30467.591} C_VEL
LIN {X 0,Y 119.669,Z 520.131,A -85,B 0,C 180,E1 -30474.036,E2 -30474.036} C_VEL
LIN {X 0,Y 124.553,Z 525.823,A -85,B 0,C 180,E1 -30480.99,E2 -30480.99} C_VEL
LIN {X 0,Y 130.224,Z 529.843,A -85,B 0,C 180,E1 -30486.554,E2 -30486.554} C_VEL
LIN {X 0,Y 138.112,Z 533.42,A -85,B 0,C 180,E1 -30492.223,E2 -30492.223} C_VEL
LIN {X 0,Y 144.967,Z 535.517,A -85,B 0,C 180,E1 -30495.972,E2 -30495.972} C_VEL
LIN {X 0,Y 156.567,Z 537.703,A -85,B 0,C 180,E1 -30500.934,E2 -30500.934} C_VEL
LIN {X 0,Y 169.645,Z 538.967,A -85,B 0,C 180,E1 -30505.247,E2 -30505.247} C_VEL
LIN {X 0,Y 184.478,Z 539.278,A -85,B 0,C 180,E1 -30509.179,E2 -30509.179} C_VEL
LIN {X 0,Y 183.407,Z 539.325,A -85,B 0,C 180,E1 -30509.303,E2 -30509.303} C_VEL
LIN {X 0,Y 182.154,Z 539.357,A -85,B 0,C 180,E1 -30509.262,E2 -30509.262} C_VEL
LIN {X 0,Y 174.997,Z 539.511,A -85,B 0,C 180,E1 -30508.438,E2 -30508.438} C_VEL
LIN {X 0,Y 165.848,Z 539.499,A -85,B 0,C 180,E1 -30506.836,E2 -30506.836} C_VEL
LIN {X 0,Y 160.897,Z 539.402,A -85,B 0,C 180,E1 -30505.726,E2 -30505.726} C_VEL
LIN {X 0,Y 156.295,Z 539.199,A -85,B 0,C 180,E1 -30504.41,E2 -30504.41} C_VEL
LIN {X 0,Y 141.268,Z 537.368,A -85,B 0,C 180,E1 -30498.522,E2 -30498.522} C_VEL
LIN {X 0,Y 131.923,Z 535.18,A -85,B 0,C 180,E1 -30493.514,E2 -30493.514} C_VEL
LIN {X 0,Y 122.42,Z 531.195,A -85,B 0,C 180,E1 -30486.306,E2 -30486.306} C_VEL
LIN {X 0,Y 116.71,Z 527.115,A -85,B 0,C 180,E1 -30479.965,E2 -30479.965} C_VEL
LIN {X 0,Y 113.036,Z 522.713,A -85,B 0,C 180,E1 -30473.924,E2 -30473.924} C_VEL
LIN {X 0,Y 110.597,Z 516.838,A -85,B 0,C 180,E1 -30466.946,E2 -30466.946} C_VEL
LIN {X 0,Y 109.889,Z 509.66,A -85,B 0,C 180,E1 -30459.756,E2 -30459.756} C_VEL
LIN {X 0,Y 110.608,Z 502.501,A -85,B 0,C 180,E1 -30453.773,E2 -30453.773} C_VEL
LIN {X 0,Y 112.088,Z 495.194,A -85,B 0,C 180,E1 -30448.624,E2 -30448.624} C_VEL
LIN {X 0,Y 113.919,Z 488.06,A -85,B 0,C 180,E1 -30444.361,E2 -30444.361} C_VEL
LIN {X 0,Y 116.241,Z 479.493,A -85,B 0,C 180,E1 -30440.022,E2 -30440.022} C_VEL
LIN {X 0,Y 118.712,Z 469.915,A -85,B 0,C 180,E1 -30435.889,E2 -30435.889} C_VEL
LIN {X 0,Y 119.499,Z 465.527,A -85,B 0,C 180,E1 -30433.604,E2 -30433.604} C_VEL
LIN {X 0,Y 119.919,Z 461.773,A -85,B 0,C 180,E1 -30431.135,E2 -30431.135} C_VEL
LIN {X 0,Y 120.058,Z 458.272,A -85,B 0,C 180,E1 -30427.897,E2 -30427.897} C_VEL
LIN {X 0,Y 120.122,Z 456.76,A -85,B 0,C 180,E1 -30425.958,E2 -30425.958} C_VEL
LIN {X 0,Y 120.206,Z 455.363,A -85,B 0,C 180,E1 -30423.35,E2 -30423.35} C_VEL
LIN {X 0,Y 120.46,Z 454.078,A -85,B 0,C 180,E1 -30419.998,E2 -30419.998} C_VEL
LIN {X 0,Y 120.287,Z 455.509,A -85,B 0,C 180,E1 -30416.649,E2 -30416.649} C_VEL
LIN {X 0,Y 119.716,Z 457.309,A -85,B 0,C 180,E1 -30416.348,E2 -30416.348} C_VEL
LIN {X 0,Y 116.126,Z 467.182,A -85,B 0,C 180,E1 -30416.073,E2 -30416.073} C_VEL
LIN {X 0,Y 111.005,Z 478.078,A -85,B 0,C 180,E1 -30415.669,E2 -30415.669} C_VEL
LIN {X 0,Y 105.788,Z 487.066,A -85,B 0,C 180,E1 -30415.205,E2 -30415.205} C_VEL
LIN {X 0,Y 99.72,Z 495.788,A -85,B 0,C 180,E1 -30414.543,E2 -30414.543} C_VEL
LIN {X 0,Y 93.66,Z 503.175,A -85,B 0,C 180,E1 -30413.837,E2 -30413.837} C_VEL
LIN {X 0,Y 86.761,Z 510.387,A -85,B 0,C 180,E1 -30412.875,E2 -30412.875} C_VEL
LIN {X 0,Y 79.895,Z 516.583,A -85,B 0,C 180,E1 -30411.724,E2 -30411.724} C_VEL
LIN {X 0,Y 71.375,Z 523.116,A -85,B 0,C 180,E1 -30409.944,E2 -30409.944} C_VEL
LIN {X 0,Y 62.795,Z 528.671,A -85,B 0,C 180,E1 -30407.547,E2 -30407.547} C_VEL
LIN {X 0,Y 54.705,Z 533.112,A -85,B 0,C 180,E1 -30404.475,E2 -30404.475} C_VEL
LIN {X 0,Y 45.012,Z 537.438,A -85,B 0,C 180,E1 -30399.518,E2 -30399.518} C_VEL
LIN {X 0,Y 38.84,Z 539.809,A -85,B 0,C 180,E1 -30394.785,E2 -30394.785} C_VEL
LIN {X 0,Y 32.989,Z 541.612,A -85,B 0,C 180,E1 -30388.446,E2 -30388.446} C_VEL
LIN {X 0,Y 23.507,Z 544.079,A -85,B 0,C 180,E1 -30366.723,E2 -30366.723} C_VEL
LIN {X 0,Y 20.711,Z 544.68,A -85,B 0,C 180,E1 -30349.836,E2 -30349.836} C_VEL
LIN {X 0,Y 19.98,Z 544.846,A -85,B 0,C 180,E1 -30330,E2 -30330} C_VEL
LIN {X 0,Y 20.753,Z 544.681,A -85,B 0,C 180,E1 -30310.206,E2 -30310.206} C_VEL
LIN {X 0,Y 23.514,Z 544.08,A -85,B 0,C 180,E1 -30293.29,E2 -30293.29} C_VEL
LIN {X 0,Y 32.989,Z 541.612,A -85,B 0,C 180,E1 -30271.554,E2 -30271.554} C_VEL
LIN {X 0,Y 41.903,Z 538.657,A -85,B 0,C 180,E1 -30262.715,E2 -30262.715} C_VEL
LIN {X 0,Y 51.445,Z 534.667,A -85,B 0,C 180,E1 -30257.007,E2 -30257.007} C_VEL
LIN {X 0,Y 61.277,Z 529.534,A -85,B 0,C 180,E1 -30252.891,E2 -30252.891} C_VEL
LIN {X 0,Y 69.679,Z 524.271,A -85,B 0,C 180,E1 -30250.459,E2 -30250.459} C_VEL
LIN {X 0,Y 78.181,Z 517.958,A -85,B 0,C 180,E1 -30248.582,E2 -30248.582} C_VEL
LIN {X 0,Y 85.04,Z 512.012,A -85,B 0,C 180,E1 -30247.389,E2 -30247.389} C_VEL
LIN {X 0,Y 91.924,Z 505.09,A -85,B 0,C 180,E1 -30246.341,E2 -30246.341} C_VEL
LIN {X 0,Y 98.849,Z 496.92,A -85,B 0,C 180,E1 -30245.527,E2 -30245.527} C_VEL
LIN {X 0,Y 104.922,Z 488.418,A -85,B 0,C 180,E1 -30244.9,E2 -30244.9} C_VEL
LIN {X 0,Y 110.139,Z 479.71,A -85,B 0,C 180,E1 -30244.43,E2 -30244.43} C_VEL
LIN {X 0,Y 114.875,Z 470.08,A -85,B 0,C 180,E1 -30244.047,E2 -30244.047} C_VEL
LIN {X 0,Y 118.62,Z 460.553,A -85,B 0,C 180,E1 -30243.749,E2 -30243.749} C_VEL
LIN {X 0,Y 119.716,Z 457.309,A -85,B 0,C 180,E1 -30243.649,E2 -30243.649} C_VEL
LIN {X 0,Y 120.288,Z 455.506,A -85,B 0,C 180,E1 -30243.351,E2 -30243.351} C_VEL
LIN {X 0,Y 120.466,Z 454.056,A -85,B 0,C 180,E1 -30240.002,E2 -30240.002} C_VEL
LIN {X 0,Y 120.213,Z 455.344,A -85,B 0,C 180,E1 -30236.65,E2 -30236.65} C_VEL
LIN {X 0,Y 120.109,Z 457.27,A -85,B 0,C 180,E1 -30233.281,E2 -30233.281} C_VEL
LIN {X 0,Y 120.061,Z 458.682,A -85,B 0,C 180,E1 -30231.587,E2 -30231.587} C_VEL
LIN {X 0,Y 119.842,Z 463.18,A -85,B 0,C 180,E1 -30227.844,E2 -30227.844} C_VEL
LIN {X 0,Y 119.251,Z 467.07,A -85,B 0,C 180,E1 -30225.497,E2 -30225.497} C_VEL
LIN {X 0,Y 118.228,Z 472.199,A -85,B 0,C 180,E1 -30223.157,E2 -30223.157} C_VEL
LIN {X 0,Y 115.474,Z 482.472,A -85,B 0,C 180,E1 -30218.584,E2 -30218.584} C_VEL
